LIN {X 0,Y 560.562,Z 1121.006,A -85,B 0,C 180,E1 21527.974,E2 21527.974} C_VEL
LIN {X 0,Y 560.296,Z 1132.318,A -85,B 0,C 180,E1 21525.845,E2 21525.845} C_VEL
LIN {X 0,Y 560.127,Z 1141.995,A -85,B 0,C 180,E1 21523.734,E2 21523.734} C_VEL
LIN {X 0,Y 560.015,Z 1150.716,A -85,B 0,C 180,E1 21521.425,E2 21521.425} C_VEL
LIN {X 0,Y 559.955,Z 1157.475,A -85,B 0,C 180,E1 21519.248,E2 21519.248} C_VEL
LIN {X 0,Y 559.899,Z 1162.84,A -85,B 0,C 180,E1 21516.975,E2 21516.975} C_VEL
LIN {X 0,Y 559.906,Z 1166.595,A -85,B 0,C 180,E1 21514.815,E2 21514.815} C_VEL
LIN {X 0,Y 559.915,Z 1169.055,A -85,B 0,C 180,E1 21512.456,E2 21512.456} C_VEL
LIN {X 0,Y 559.892,Z 1169.939,A -85,B 0,C 180,E1 21510.307,E2 21510.307} C_VEL
LIN {X 0,Y 559.911,Z 1169.324,A -85,B 0,C 180,E1 21507.953,E2 21507.953} C_VEL
LIN {X 0,Y 559.914,Z 1167.276,A -85,B 0,C 180,E1 21505.699,E2 21505.699} C_VEL
LIN {X 0,Y 559.914,Z 1163.461,A -85,B 0,C 180,E1 21503.334,E2 21503.334} C_VEL
LIN {X 0,Y 559.955,Z 1158.551,A -85,B 0,C 180,E1 21501.167,E2 21501.167} C_VEL
LIN {X 0,Y 560,Z 1151.764,A -85,B 0,C 180,E1 21498.882,E2 21498.882} C_VEL
LIN {X 0,Y 560.097,Z 1144.109,A -85,B 0,C 180,E1 21496.791,E2 21496.791} C_VEL
LIN {X 0,Y 560.276,Z 1133.883,A -85,B 0,C 180,E1 21494.473,E2 21494.473} C_VEL
LIN {X 0,Y 560.534,Z 1122.819,A -85,B 0,C 180,E1 21492.348,E2 21492.348} C_VEL
LIN {X 0,Y 560.864,Z 1109.753,A -85,B 0,C 180,E1 21490.201,E2 21490.201} C_VEL
LIN {X 0,Y 561.293,Z 1095.338,A -85,B 0,C 180,E1 21488.137,E2 21488.137} C_VEL
LIN {X 0,Y 561.795,Z 1079.942,A -85,B 0,C 180,E1 21486.227,E2 21486.227} C_VEL
LIN {X 0,Y 562.438,Z 1062.115,A -85,B 0,C 180,E1 21484.293,E2 21484.293} C_VEL
LIN {X 0,Y 563.12,Z 1044.253,A -85,B 0,C 180,E1 21482.595,E2 21482.595} C_VEL
LIN {X 0,Y 563.844,Z 1025.338,A -85,B 0,C 180,E1 21481.046,E2 21481.046} C_VEL
LIN {X 0,Y 564.61,Z 1004.603,A -85,B 0,C 180,E1 21479.571,E2 21479.571} C_VEL
LIN {X 0,Y 565.354,Z 984.83,A -85,B 0,C 180,E1 21478.374,E2 21478.374} C_VEL
LIN {X 0,Y 566.073,Z 962.172,A -85,B 0,C 180,E1 21477.22,E2 21477.22} C_VEL
LIN {X 0,Y 566.732,Z 941.505,A -85,B 0,C 180,E1 21476.36,E2 21476.36} C_VEL
LIN {X 0,Y 567.278,Z 918.342,A -85,B 0,C 180,E1 21475.6,E2 21475.6} C_VEL
LIN {X 0,Y 567.741,Z 896.292,A -85,B 0,C 180,E1 21475.062,E2 21475.062} C_VEL
LIN {X 0,Y 568.079,Z 859.915,A -85,B 0,C 180,E1 21474.482,E2 21474.482} C_VEL
LIN {X 0,Y 569.548,Z 649.859,A -85,B 0,C 180,E1 21471.336,E2 21471.336} C_VEL
LIN {X 0,Y 570.107,Z 551.64,A -85,B 0,C 180,E1 21469.813,E2 21469.813} C_VEL
LIN {X 0,Y 568.373,Z 542.27,A -85,B 0,C 180,E1 21469.502,E2 21469.502} C_VEL
LIN {X 0,Y 568.462,Z 530.87,A -85,B 0,C 180,E1 21468.749,E2 21468.749} C_VEL
LIN {X 0,Y 561.578,Z 516.737,A -85,B 0,C 180,E1 21467.146,E2 21467.146} C_VEL
LIN {X 0,Y 560.294,Z 513.438,A -85,B 0,C 180,E1 21466.726,E2 21466.726} C_VEL
LIN {X 0,Y 560.28,Z 513.252,A -85,B 0,C 180,E1 21463.397,E2 21463.397} C_VEL
LIN {X 0,Y 560.273,Z 513.252,A -85,B 0,C 180,E1 21459.975,E2 21459.975} C_VEL
LIN {X 0,Y 560.264,Z 513.243,A -85,B 0,C 180,E1 21456.715,E2 21456.715} C_VEL
LIN {X 0,Y 560.267,Z 513.249,A -85,B 0,C 180,E1 21453.466,E2 21453.466} C_VEL
LIN {X 0,Y 560.261,Z 513.255,A -85,B 0,C 180,E1 21450.216,E2 21450.216} C_VEL
LIN {X 0,Y 560.264,Z 513.249,A -85,B 0,C 180,E1 21446.955,E2 21446.955} C_VEL
LIN {X 0,Y 560.265,Z 513.258,A -85,B 0,C 180,E1 21443.674,E2 21443.674} C_VEL
LIN {X 0,Y 560.269,Z 513.249,A -85,B 0,C 180,E1 21440.365,E2 21440.365} C_VEL
LIN {X 0,Y 560.277,Z 513.251,A -85,B 0,C 180,E1 21436.911,E2 21436.911} C_VEL
LIN {X 0,Y 560.27,Z 513.247,A -85,B 0,C 180,E1 21433.52,E2 21433.52} C_VEL
LIN {X 0,Y 560.262,Z 513.247,A -85,B 0,C 180,E1 21430.176,E2 21430.176} C_VEL
LIN {X 0,Y 560.264,Z 513.248,A -85,B 0,C 180,E1 21426.867,E2 21426.867} C_VEL
LIN {X 0,Y 560.263,Z 513.25,A -85,B 0,C 180,E1 21423.581,E2 21423.581} C_VEL
LIN {X 0,Y 560.277,Z 513.258,A -85,B 0,C 180,E1 21420.204,E2 21420.204} C_VEL
LIN {X 0,Y 560.278,Z 513.25,A -85,B 0,C 180,E1 21416.726,E2 21416.726} C_VEL
LIN {X 0,Y 560.261,Z 513.254,A -85,B 0,C 180,E1 21413.338,E2 21413.338} C_VEL
LIN {X 0,Y 560.268,Z 513.255,A -85,B 0,C 180,E1 21410.031,E2 21410.031} C_VEL
LIN {X 0,Y 560.258,Z 513.247,A -85,B 0,C 180,E1 21406.795,E2 21406.795} C_VEL
LIN {X 0,Y 560.27,Z 513.258,A -85,B 0,C 180,E1 21403.516,E2 21403.516} C_VEL
LIN {X 0,Y 560.264,Z 513.244,A -85,B 0,C 180,E1 21400.179,E2 21400.179} C_VEL
LIN {X 0,Y 560.278,Z 513.256,A -85,B 0,C 180,E1 21396.772,E2 21396.772} C_VEL
LIN {X 0,Y 560.255,Z 513.251,A -85,B 0,C 180,E1 21396.282,E2 21396.282} C_VEL
LIN {X 0,Y 559.277,Z 513.372,A -85,B 0,C 180,E1 21395.494,E2 21395.494} C_VEL
LIN {X 0,Y 552.874,Z 514.168,A -85,B 0,C 180,E1 21393.282,E2 21393.282} C_VEL
LIN {X 0,Y 552.338,Z 514.243,A -85,B 0,C 180,E1 21392.706,E2 21392.706} C_VEL
LIN {X 0,Y 552.341,Z 514.229,A -85,B 0,C 180,E1 21389.301,E2 21389.301} C_VEL
LIN {X 0,Y 552.324,Z 514.245,A -85,B 0,C 180,E1 21385.987,E2 21385.987} C_VEL
LIN {X 0,Y 552.334,Z 514.241,A -85,B 0,C 180,E1 21382.627,E2 21382.627} C_VEL
LIN {X 0,Y 552.314,Z 514.238,A -85,B 0,C 180,E1 21379.329,E2 21379.329} C_VEL
LIN {X 0,Y 552.335,Z 514.233,A -85,B 0,C 180,E1 21375.962,E2 21375.962} C_VEL
LIN {X 0,Y 552.323,Z 514.225,A -85,B 0,C 180,E1 21372.613,E2 21372.613} C_VEL
LIN {X 0,Y 552.388,Z 514.576,A -85,B 0,C 180,E1 21371.593,E2 21371.593} C_VEL
LIN {X 0,Y 554.03,Z 518.332,A -85,B 0,C 180,E1 21371.109,E2 21371.109} C_VEL
LIN {X 0,Y 560.868,Z 533.617,A -85,B 0,C 180,E1 21369.368,E2 21369.368} C_VEL
LIN {X 0,Y 559.531,Z 581.004,A -85,B 0,C 180,E1 21366.127,E2 21366.127} C_VEL
LIN {X 0,Y 559.41,Z 590.555,A -85,B 0,C 180,E1 21365.522,E2 21365.522} C_VEL
LIN {X 0,Y 561.19,Z 601.495,A -85,B 0,C 180,E1 21365.221,E2 21365.221} C_VEL
LIN {X 0,Y 559.53,Z 831.551,A -85,B 0,C 180,E1 21361.866,E2 21361.866} C_VEL
LIN {X 0,Y 559.039,Z 897.029,A -85,B 0,C 180,E1 21360.896,E2 21360.896} C_VEL
LIN {X 0,Y 558.577,Z 918.635,A -85,B 0,C 180,E1 21360.381,E2 21360.381} C_VEL
LIN {X 0,Y 558.024,Z 940.668,A -85,B 0,C 180,E1 21359.655,E2 21359.655} C_VEL
LIN {X 0,Y 557.432,Z 961.155,A -85,B 0,C 180,E1 21358.79,E2 21358.79} C_VEL
LIN {X 0,Y 556.733,Z 980.474,A -85,B 0,C 180,E1 21357.778,E2 21357.778} C_VEL
LIN {X 0,Y 555.975,Z 1001.01,A -85,B 0,C 180,E1 21356.487,E2 21356.487} C_VEL
LIN {X 0,Y 555.267,Z 1019.082,A -85,B 0,C 180,E1 21355.148,E2 21355.148} C_VEL
LIN {X 0,Y 554.564,Z 1036.919,A -85,B 0,C 180,E1 21353.594,E2 21353.594} C_VEL
LIN {X 0,Y 553.926,Z 1053.575,A -85,B 0,C 180,E1 21351.907,E2 21351.907} C_VEL
LIN {X 0,Y 553.35,Z 1069.662,A -85,B 0,C 180,E1 21350.016,E2 21350.016} C_VEL
LIN {X 0,Y 552.9,Z 1083.542,A -85,B 0,C 180,E1 21348.122,E2 21348.122} C_VEL
LIN {X 0,Y 552.547,Z 1095.699,A -85,B 0,C 180,E1 21346.181,E2 21346.181} C_VEL
LIN {X 0,Y 552.274,Z 1107.096,A -85,B 0,C 180,E1 21344.04,E2 21344.04} C_VEL
LIN {X 0,Y 552.098,Z 1116.58,A -85,B 0,C 180,E1 21341.915,E2 21341.915} C_VEL
LIN {X 0,Y 551.991,Z 1124.218,A -85,B 0,C 180,E1 21339.808,E2 21339.808} C_VEL
LIN {X 0,Y 551.933,Z 1130.536,A -85,B 0,C 180,E1 21337.599,E2 21337.599} C_VEL
LIN {X 0,Y 551.913,Z 1135.247,A -85,B 0,C 180,E1 21335.406,E2 21335.406} C_VEL
LIN {X 0,Y 551.909,Z 1138.236,A -85,B 0,C 180,E1 21333.219,E2 21333.219} C_VEL
LIN {X 0,Y 551.906,Z 1139.795,A -85,B 0,C 180,E1 21330.934,E2 21330.934} C_VEL
LIN {X 0,Y 551.91,Z 1139.747,A -85,B 0,C 180,E1 21328.754,E2 21328.754} C_VEL
LIN {X 0,Y 551.914,Z 1138.102,A -85,B 0,C 180,E1 21326.566,E2 21326.566} C_VEL
LIN {X 0,Y 551.922,Z 1135.016,A -85,B 0,C 180,E1 21324.386,E2 21324.386} C_VEL
LIN {X 0,Y 551.936,Z 1130.443,A -85,B 0,C 180,E1 21322.272,E2 21322.272} C_VEL
LIN {X 0,Y 551.999,Z 1123.827,A -85,B 0,C 180,E1 21319.986,E2 21319.986} C_VEL
LIN {X 0,Y 552.112,Z 1116.11,A -85,B 0,C 180,E1 21317.873,E2 21317.873} C_VEL
LIN {X 0,Y 552.292,Z 1106.494,A -85,B 0,C 180,E1 21315.746,E2 21315.746} C_VEL
LIN {X 0,Y 552.57,Z 1094.958,A -85,B 0,C 180,E1 21313.604,E2 21313.604} C_VEL
LIN {X 0,Y 552.928,Z 1082.692,A -85,B 0,C 180,E1 21311.661,E2 21311.661} C_VEL
LIN {X 0,Y 553.372,Z 1069.014,A -85,B 0,C 180,E1 21309.811,E2 21309.811} C_VEL
LIN {X 0,Y 553.947,Z 1053.078,A -85,B 0,C 180,E1 21307.949,E2 21307.949} C_VEL
LIN {X 0,Y 554.603,Z 1035.953,A -85,B 0,C 180,E1 21306.227,E2 21306.227} C_VEL
LIN {X 0,Y 555.316,Z 1017.95,A -85,B 0,C 180,E1 21304.671,E2 21304.671} C_VEL
LIN {X 0,Y 556.05,Z 999.031,A -85,B 0,C 180,E1 21303.286,E2 21303.286} C_VEL
LIN {X 0,Y 556.788,Z 979.033,A -85,B 0,C 180,E1 21302.05,E2 21302.05} C_VEL
LIN {X 0,Y 557.472,Z 959.341,A -85,B 0,C 180,E1 21301.036,E2 21301.036} C_VEL
LIN {X 0,Y 558.068,Z 939.628,A -85,B 0,C 180,E1 21300.216,E2 21300.216} C_VEL
LIN {X 0,Y 558.594,Z 917.254,A -85,B 0,C 180,E1 21299.491,E2 21299.491} C_VEL
LIN {X 0,Y 559.054,Z 895.666,A -85,B 0,C 180,E1 21298.991,E2 21298.991} C_VEL
LIN {X 0,Y 560.624,Z 674.56,A -85,B 0,C 180,E1 21295.764,E2 21295.764} C_VEL
LIN {X 0,Y 560.976,Z 601.536,A -85,B 0,C 180,E1 21294.674,E2 21294.674} C_VEL
LIN {X 0,Y 558.666,Z 590.554,A -85,B 0,C 180,E1 21294.306,E2 21294.306} C_VEL
LIN {X 0,Y 559.886,Z 549.146,A -85,B 0,C 180,E1 21290.92,E2 21290.92} C_VEL
LIN {X 0,Y 560.191,Z 533.38,A -85,B 0,C 180,E1 21289.574,E2 21289.574} C_VEL
LIN {X 0,Y 553.416,Z 517.359,A -85,B 0,C 180,E1 21287.488,E2 21287.488} C_VEL
LIN {X 0,Y 552.342,Z 514.443,A -85,B 0,C 180,E1 21287.064,E2 21287.064} C_VEL
LIN {X 0,Y 552.283,Z 514.237,A -85,B 0,C 180,E1 21284.043,E2 21284.043} C_VEL
LIN {X 0,Y 552.303,Z 514.239,A -85,B 0,C 180,E1 21280.665,E2 21280.665} C_VEL
LIN {X 0,Y 552.28,Z 514.249,A -85,B 0,C 180,E1 21277.706,E2 21277.706} C_VEL
LIN {X 0,Y 552.336,Z 514.514,A -85,B 0,C 180,E1 21275.33,E2 21275.33} C_VEL
LIN {X 0,Y 556.826,Z 528.593,A -85,B 0,C 180,E1 21273.943,E2 21273.943} C_VEL
LIN {X 0,Y 556.497,Z 566.554,A -85,B 0,C 180,E1 21271.015,E2 21271.015} C_VEL
LIN {X 0,Y 555.991,Z 605.609,A -85,B 0,C 180,E1 21267.993,E2 21267.993} C_VEL
LIN {X 0,Y 555.136,Z 647.932,A -85,B 0,C 180,E1 21264.7,E2 21264.7} C_VEL
LIN {X 0,Y 554.341,Z 692.274,A -85,B 0,C 180,E1 21261.312,E2 21261.312} C_VEL
LIN {X 0,Y 554.138,Z 705.669,A -85,B 0,C 180,E1 21260.336,E2 21260.336} C_VEL
LIN {X 0,Y 554.992,Z 713.85,A -85,B 0,C 180,E1 21260.192,E2 21260.192} C_VEL
LIN {X 0,Y 554.361,Z 876.056,A -85,B 0,C 180,E1 21258.008,E2 21258.008} C_VEL
LIN {X 0,Y 554.144,Z 893.538,A -85,B 0,C 180,E1 21257.571,E2 21257.571} C_VEL
LIN {X 0,Y 553.859,Z 910.683,A -85,B 0,C 180,E1 21256.946,E2 21256.946} C_VEL
LIN {X 0,Y 553.556,Z 926.795,A -85,B 0,C 180,E1 21256.151,E2 21256.151} C_VEL
LIN {X 0,Y 553.207,Z 942.641,A -85,B 0,C 180,E1 21255.145,E2 21255.145} C_VEL
LIN {X 0,Y 552.864,Z 957.964,A -85,B 0,C 180,E1 21253.918,E2 21253.918} C_VEL
LIN {X 0,Y 552.575,Z 970.819,A -85,B 0,C 180,E1 21252.647,E2 21252.647} C_VEL
LIN {X 0,Y 552.341,Z 982.209,A -85,B 0,C 180,E1 21251.274,E2 21251.274} C_VEL
LIN {X 0,Y 552.158,Z 992.869,A -85,B 0,C 180,E1 21249.695,E2 21249.695} C_VEL
LIN {X 0,Y 552.03,Z 1001.869,A -85,B 0,C 180,E1 21248.017,E2 21248.017} C_VEL
LIN {X 0,Y 551.96,Z 1008.816,A -85,B 0,C 180,E1 21246.344,E2 21246.344} C_VEL
LIN {X 0,Y 551.925,Z 1014.226,A -85,B 0,C 180,E1 21244.572,E2 21244.572} C_VEL
LIN {X 0,Y 551.915,Z 1017.967,A -85,B 0,C 180,E1 21242.7,E2 21242.7} C_VEL
LIN {X 0,Y 551.914,Z 1019.781,A -85,B 0,C 180,E1 21240.831,E2 21240.831} C_VEL
LIN {X 0,Y 551.915,Z 1019.746,A -85,B 0,C 180,E1 21239.066,E2 21239.066} C_VEL
LIN {X 0,Y 551.915,Z 1018.103,A -85,B 0,C 180,E1 21237.301,E2 21237.301} C_VEL
LIN {X 0,Y 551.925,Z 1014.451,A -85,B 0,C 180,E1 21235.428,E2 21235.428} C_VEL
LIN {X 0,Y 551.955,Z 1009.461,A -85,B 0,C 180,E1 21233.761,E2 21233.761} C_VEL
LIN {X 0,Y 552.02,Z 1002.789,A -85,B 0,C 180,E1 21232.088,E2 21232.088} C_VEL
LIN {X 0,Y 552.14,Z 994.047,A -85,B 0,C 180,E1 21230.41,E2 21230.41} C_VEL
LIN {X 0,Y 552.317,Z 983.658,A -85,B 0,C 180,E1 21228.831,E2 21228.831} C_VEL
LIN {X 0,Y 552.564,Z 971.117,A -85,B 0,C 180,E1 21227.3,E2 21227.3} C_VEL
LIN {X 0,Y 552.818,Z 959.469,A -85,B 0,C 180,E1 21226.135,E2 21226.135} C_VEL
LIN {X 0,Y 553.134,Z 946.112,A -85,B 0,C 180,E1 21225.02,E2 21225.02} C_VEL
LIN {X 0,Y 553.47,Z 930.113,A -85,B 0,C 180,E1 21223.955,E2 21223.955} C_VEL
LIN {X 0,Y 553.749,Z 915.956,A -85,B 0,C 180,E1 21223.208,E2 21223.208} C_VEL
LIN {X 0,Y 554.051,Z 900.589,A -85,B 0,C 180,E1 21222.569,E2 21222.569} C_VEL
LIN {X 0,Y 554.278,Z 883.504,A -85,B 0,C 180,E1 21222.066,E2 21222.066} C_VEL
LIN {X 0,Y 554.42,Z 865.876,A -85,B 0,C 180,E1 21221.739,E2 21221.739} C_VEL
LIN {X 0,Y 554.815,Z 710.464,A -85,B 0,C 180,E1 21219.665,E2 21219.665} C_VEL
LIN {X 0,Y 554.077,Z 704.577,A -85,B 0,C 180,E1 21219.522,E2 21219.522} C_VEL
LIN {X 0,Y 554.903,Z 660.003,A -85,B 0,C 180,E1 21216.139,E2 21216.139} C_VEL
LIN {X 0,Y 555.761,Z 617.071,A -85,B 0,C 180,E1 21212.809,E2 21212.809} C_VEL
LIN {X 0,Y 556.004,Z 585.332,A -85,B 0,C 180,E1 21210.438,E2 21210.438} C_VEL
LIN {X 0,Y 555.825,Z 557.018,A -85,B 0,C 180,E1 21208.435,E2 21208.435} C_VEL
LIN {X 0,Y 555.246,Z 527.459,A -85,B 0,C 180,E1 21206.486,E2 21206.486} C_VEL
LIN {X 0,Y 554.798,Z 524.469,A -85,B 0,C 180,E1 21206.284,E2 21206.284} C_VEL
LIN {X 0,Y 552.369,Z 514.601,A -85,B 0,C 180,E1 21205.568,E2 21205.568} C_VEL
LIN {X 0,Y 552.343,Z 514.249,A -85,B 0,C 180,E1 21205.088,E2 21205.088} C_VEL
LIN {X 0,Y 552.318,Z 514.245,A -85,B 0,C 180,E1 21201.749,E2 21201.749} C_VEL
LIN {X 0,Y 552.325,Z 514.244,A -85,B 0,C 180,E1 21198.367,E2 21198.367} C_VEL
LIN {X 0,Y 552.319,Z 514.23,A -85,B 0,C 180,E1 21195.058,E2 21195.058} C_VEL
LIN {X 0,Y 552.388,Z 514.56,A -85,B 0,C 180,E1 21194.396,E2 21194.396} C_VEL
LIN {X 0,Y 553.864,Z 518.049,A -85,B 0,C 180,E1 21193.922,E2 21193.922} C_VEL
LIN {X 0,Y 561.374,Z 535.018,A -85,B 0,C 180,E1 21191.769,E2 21191.769} C_VEL
LIN {X 0,Y 561.249,Z 543.948,A -85,B 0,C 180,E1 21191.09,E2 21191.09} C_VEL
LIN {X 0,Y 564.108,Z 557.393,A -85,B 0,C 180,E1 21190.61,E2 21190.61} C_VEL
LIN {X 0,Y 562.326,Z 765.247,A -85,B 0,C 180,E1 21187.415,E2 21187.415} C_VEL
LIN {X 0,Y 561.248,Z 892.082,A -85,B 0,C 180,E1 21185.487,E2 21185.487} C_VEL
LIN {X 0,Y 560.694,Z 915.746,A -85,B 0,C 180,E1 21184.939,E2 21184.939} C_VEL
LIN {X 0,Y 560.122,Z 937.778,A -85,B 0,C 180,E1 21184.241,E2 21184.241} C_VEL
LIN {X 0,Y 559.344,Z 959.681,A -85,B 0,C 180,E1 21183.345,E2 21183.345} C_VEL
LIN {X 0,Y 558.545,Z 980.784,A -85,B 0,C 180,E1 21182.3,E2 21182.3} C_VEL
LIN {X 0,Y 557.68,Z 1001.047,A -85,B 0,C 180,E1 21181.088,E2 21181.088} C_VEL
LIN {X 0,Y 556.795,Z 1020.931,A -85,B 0,C 180,E1 21179.711,E2 21179.711} C_VEL
LIN {X 0,Y 555.953,Z 1039.504,A -85,B 0,C 180,E1 21178.208,E2 21178.208} C_VEL
LIN {X 0,Y 555.077,Z 1058.792,A -85,B 0,C 180,E1 21176.418,E2 21176.418} C_VEL
LIN {X 0,Y 554.366,Z 1075.661,A -85,B 0,C 180,E1 21174.622,E2 21174.622} C_VEL
LIN {X 0,Y 553.688,Z 1091.994,A -85,B 0,C 180,E1 21172.621,E2 21172.621} C_VEL
LIN {X 0,Y 553.14,Z 1106.919,A -85,B 0,C 180,E1 21170.529,E2 21170.529} C_VEL
LIN {X 0,Y 552.722,Z 1119.734,A -85,B 0,C 180,E1 21168.456,E2 21168.456} C_VEL
LIN {X 0,Y 552.396,Z 1131.799,A -85,B 0,C 180,E1 21166.185,E2 21166.185} C_VEL
LIN {X 0,Y 552.203,Z 1141.076,A -85,B 0,C 180,E1 21164.149,E2 21164.149} C_VEL
LIN {X 0,Y 552.051,Z 1150.341,A -85,B 0,C 180,E1 21161.704,E2 21161.704} C_VEL
LIN {X 0,Y 551.951,Z 1156.868,A -85,B 0,C 180,E1 21159.594,E2 21159.594} C_VEL
LIN {X 0,Y 551.902,Z 1162.634,A -85,B 0,C 180,E1 21157.181,E2 21157.181} C_VEL
LIN {X 0,Y 551.913,Z 1166.276,A -85,B 0,C 180,E1 21155.093,E2 21155.093} C_VEL
LIN {X 0,Y 551.91,Z 1168.988,A -85,B 0,C 180,E1 21152.596,E2 21152.596} C_VEL
LIN {X 0,Y 551.884,Z 1169.895,A -85,B 0,C 180,E1 21150.519,E2 21150.519} C_VEL
LIN {X 0,Y 551.908,Z 1169.391,A -85,B 0,C 180,E1 21148.027,E2 21148.027} C_VEL
LIN {X 0,Y 551.917,Z 1167.503,A -85,B 0,C 180,E1 21145.844,E2 21145.844} C_VEL
LIN {X 0,Y 551.916,Z 1163.667,A -85,B 0,C 180,E1 21143.342,E2 21143.342} C_VEL
LIN {X 0,Y 551.96,Z 1159.061,A -85,B 0,C 180,E1 21141.248,E2 21141.248} C_VEL
LIN {X 0,Y 552.018,Z 1152.119,A -85,B 0,C 180,E1 21138.825,E2 21138.825} C_VEL
LIN {X 0,Y 552.129,Z 1144.519,A -85,B 0,C 180,E1 21136.704,E2 21136.704} C_VEL
LIN {X 0,Y 552.342,Z 1134.4,A -85,B 0,C 180,E1 21134.352,E2 21134.352} C_VEL
LIN {X 0,Y 552.639,Z 1123.402,A -85,B 0,C 180,E1 21132.196,E2 21132.196} C_VEL
LIN {X 0,Y 553.038,Z 1110.464,A -85,B 0,C 180,E1 21130.019,E2 21130.019} C_VEL
LIN {X 0,Y 553.551,Z 1096.068,A -85,B 0,C 180,E1 21127.912,E2 21127.912} C_VEL
LIN {X 0,Y 554.162,Z 1080.254,A -85,B 0,C 180,E1 21125.917,E2 21125.917} C_VEL
LIN {X 0,Y 554.942,Z 1062.116,A -85,B 0,C 180,E1 21123.92,E2 21123.92} C_VEL
LIN {X 0,Y 555.763,Z 1043.896,A -85,B 0,C 180,E1 21122.169,E2 21122.169} C_VEL
LIN {X 0,Y 556.617,Z 1024.907,A -85,B 0,C 180,E1 21120.599,E2 21120.599} C_VEL
LIN {X 0,Y 557.56,Z 1003.716,A -85,B 0,C 180,E1 21119.084,E2 21119.084} C_VEL
LIN {X 0,Y 558.416,Z 983.884,A -85,B 0,C 180,E1 21117.877,E2 21117.877} C_VEL
LIN {X 0,Y 559.233,Z 962.234,A -85,B 0,C 180,E1 21116.77,E2 21116.77} C_VEL
LIN {X 0,Y 559.996,Z 941.503,A -85,B 0,C 180,E1 21115.9,E2 21115.9} C_VEL
LIN {X 0,Y 560.63,Z 918.219,A -85,B 0,C 180,E1 21115.13,E2 21115.13} C_VEL
LIN {X 0,Y 561.192,Z 895.804,A -85,B 0,C 180,E1 21114.581,E2 21114.581} C_VEL
LIN {X 0,Y 561.6,Z 855.786,A -85,B 0,C 180,E1 21113.945,E2 21113.945} C_VEL
LIN {X 0,Y 563.331,Z 646.028,A -85,B 0,C 180,E1 21110.767,E2 21110.767} C_VEL
LIN {X 0,Y 563.997,Z 553.429,A -85,B 0,C 180,E1 21109.316,E2 21109.316} C_VEL
LIN {X 0,Y 561.94,Z 542.168,A -85,B 0,C 180,E1 21108.935,E2 21108.935} C_VEL
LIN {X 0,Y 561.962,Z 534.582,A -85,B 0,C 180,E1 21108.421,E2 21108.421} C_VEL
LIN {X 0,Y 553.971,Z 518.181,A -85,B 0,C 180,E1 21106.515,E2 21106.515} C_VEL
LIN {X 0,Y 552.379,Z 514.586,A -85,B 0,C 180,E1 21106.062,E2 21106.062} C_VEL
LIN {X 0,Y 552.325,Z 514.23,A -85,B 0,C 180,E1 21105.204,E2 21105.204} C_VEL
LIN {X 0,Y 552.329,Z 514.241,A -85,B 0,C 180,E1 21101.911,E2 21101.911} C_VEL
LIN {X 0,Y 552.323,Z 514.248,A -85,B 0,C 180,E1 21098.552,E2 21098.552} C_VEL
LIN {X 0,Y 552.331,Z 514.245,A -85,B 0,C 180,E1 21095.271,E2 21095.271} C_VEL
LIN {X 0,Y 552.332,Z 514.234,A -85,B 0,C 180,E1 21091.896,E2 21091.896} C_VEL
LIN {X 0,Y 552.336,Z 514.238,A -85,B 0,C 180,E1 21088.43,E2 21088.43} C_VEL
LIN {X 0,Y 552.328,Z 514.248,A -85,B 0,C 180,E1 21085.062,E2 21085.062} C_VEL
LIN {X 0,Y 552.325,Z 514.232,A -85,B 0,C 180,E1 21081.771,E2 21081.771} C_VEL
LIN {X 0,Y 552.327,Z 514.244,A -85,B 0,C 180,E1 21078.453,E2 21078.453} C_VEL
LIN {X 0,Y 552.328,Z 514.23,A -85,B 0,C 180,E1 21075.11,E2 21075.11} C_VEL
LIN {X 0,Y 552.339,Z 514.24,A -85,B 0,C 180,E1 21071.668,E2 21071.668} C_VEL
LIN {X 0,Y 552.326,Z 514.232,A -85,B 0,C 180,E1 21068.222,E2 21068.222} C_VEL
LIN {X 0,Y 552.328,Z 514.244,A -85,B 0,C 180,E1 21064.88,E2 21064.88} C_VEL
LIN {X 0,Y 552.322,Z 514.244,A -85,B 0,C 180,E1 21061.556,E2 21061.556} C_VEL
LIN {X 0,Y 552.331,Z 514.246,A -85,B 0,C 180,E1 21058.236,E2 21058.236} C_VEL
LIN {X 0,Y 552.336,Z 514.24,A -85,B 0,C 180,E1 21054.807,E2 21054.807} C_VEL
LIN {X 0,Y 552.328,Z 514.248,A -85,B 0,C 180,E1 21051.358,E2 21051.358} C_VEL
LIN {X 0,Y 552.33,Z 514.234,A -85,B 0,C 180,E1 21047.984,E2 21047.984} C_VEL
LIN {X 0,Y 552.318,Z 514.245,A -85,B 0,C 180,E1 21044.674,E2 21044.674} C_VEL
LIN {X 0,Y 552.333,Z 514.234,A -85,B 0,C 180,E1 21041.312,E2 21041.312} C_VEL
LIN {X 0,Y 552.338,Z 514.241,A -85,B 0,C 180,E1 21037.881,E2 21037.881} C_VEL
LIN {X 0,Y 552.326,Z 514.234,A -85,B 0,C 180,E1 21034.479,E2 21034.479} C_VEL
LIN {X 0,Y 552.338,Z 514.243,A -85,B 0,C 180,E1 21032.706,E2 21032.706} C_VEL
LIN {X 0,Y 551.35,Z 514.375,A -85,B 0,C 180,E1 21031.907,E2 21031.907} C_VEL
LIN {X 0,Y 544.847,Z 515.163,A -85,B 0,C 180,E1 21029.605,E2 21029.605} C_VEL
LIN {X 0,Y 544.396,Z 515.217,A -85,B 0,C 180,E1 21029.079,E2 21029.079} C_VEL
LIN {X 0,Y 544.377,Z 515.231,A -85,B 0,C 180,E1 21025.743,E2 21025.743} C_VEL
LIN {X 0,Y 544.394,Z 515.232,A -85,B 0,C 180,E1 21022.427,E2 21022.427} C_VEL
LIN {X 0,Y 544.377,Z 515.227,A -85,B 0,C 180,E1 21019.166,E2 21019.166} C_VEL
LIN {X 0,Y 544.399,Z 515.219,A -85,B 0,C 180,E1 21015.739,E2 21015.739} C_VEL
LIN {X 0,Y 544.413,Z 515.335,A -85,B 0,C 180,E1 21012.379,E2 21012.379} C_VEL
LIN {X 0,Y 544.535,Z 515.993,A -85,B 0,C 180,E1 21012.225,E2 21012.225} C_VEL
LIN {X 0,Y 552.88,Z 534.192,A -85,B 0,C 180,E1 21010.014,E2 21010.014} C_VEL
LIN {X 0,Y 554.194,Z 537.39,A -85,B 0,C 180,E1 21009.66,E2 21009.66} C_VEL
LIN {X 0,Y 552.65,Z 584.849,A -85,B 0,C 180,E1 21006.38,E2 21006.38} C_VEL
LIN {X 0,Y 552.626,Z 590.599,A -85,B 0,C 180,E1 21006.026,E2 21006.026} C_VEL
LIN {X 0,Y 554.645,Z 602.933,A -85,B 0,C 180,E1 21005.678,E2 21005.678} C_VEL
LIN {X 0,Y 552.725,Z 833.51,A -85,B 0,C 180,E1 21002.277,E2 21002.277} C_VEL
LIN {X 0,Y 552.172,Z 897.066,A -85,B 0,C 180,E1 21001.323,E2 21001.323} C_VEL
LIN {X 0,Y 551.641,Z 918.695,A -85,B 0,C 180,E1 21000.803,E2 21000.803} C_VEL
LIN {X 0,Y 551.032,Z 940.353,A -85,B 0,C 180,E1 21000.084,E2 21000.084} C_VEL
LIN {X 0,Y 550.352,Z 959.947,A -85,B 0,C 180,E1 20999.256,E2 20999.256} C_VEL
LIN {X 0,Y 549.571,Z 979.496,A -85,B 0,C 180,E1 20998.231,E2 20998.231} C_VEL
LIN {X 0,Y 548.683,Z 1000.206,A -85,B 0,C 180,E1 20996.926,E2 20996.926} C_VEL
LIN {X 0,Y 547.838,Z 1019.088,A -85,B 0,C 180,E1 20995.514,E2 20995.514} C_VEL
LIN {X 0,Y 547.022,Z 1036.928,A -85,B 0,C 180,E1 20993.94,E2 20993.94} C_VEL
LIN {X 0,Y 546.285,Z 1053.274,A -85,B 0,C 180,E1 20992.264,E2 20992.264} C_VEL
LIN {X 0,Y 545.616,Z 1069.179,A -85,B 0,C 180,E1 20990.376,E2 20990.376} C_VEL
LIN {X 0,Y 545.109,Z 1082.828,A -85,B 0,C 180,E1 20988.501,E2 20988.501} C_VEL
LIN {X 0,Y 544.672,Z 1095.701,A -85,B 0,C 180,E1 20986.421,E2 20986.421} C_VEL
LIN {X 0,Y 544.349,Z 1107.1,A -85,B 0,C 180,E1 20984.249,E2 20984.249} C_VEL
LIN {X 0,Y 544.139,Z 1116.583,A -85,B 0,C 180,E1 20982.092,E2 20982.092} C_VEL
LIN {X 0,Y 544.013,Z 1124.234,A -85,B 0,C 180,E1 20979.949,E2 20979.949} C_VEL
LIN {X 0,Y 543.945,Z 1130.538,A -85,B 0,C 180,E1 20977.712,E2 20977.712} C_VEL
LIN {X 0,Y 543.918,Z 1135.248,A -85,B 0,C 180,E1 20975.485,E2 20975.485} C_VEL
LIN {X 0,Y 543.911,Z 1138.237,A -85,B 0,C 180,E1 20973.267,E2 20973.267} C_VEL
LIN {X 0,Y 543.907,Z 1139.795,A -85,B 0,C 180,E1 20970.948,E2 20970.948} C_VEL
LIN {X 0,Y 543.909,Z 1139.747,A -85,B 0,C 180,E1 20968.736,E2 20968.736} C_VEL
LIN {X 0,Y 543.912,Z 1138.109,A -85,B 0,C 180,E1 20966.522,E2 20966.522} C_VEL
LIN {X 0,Y 543.926,Z 1135.015,A -85,B 0,C 180,E1 20964.303,E2 20964.303} C_VEL
LIN {X 0,Y 543.945,Z 1130.498,A -85,B 0,C 180,E1 20962.182,E2 20962.182} C_VEL
LIN {X 0,Y 544.023,Z 1123.825,A -85,B 0,C 180,E1 20959.838,E2 20959.838} C_VEL
LIN {X 0,Y 544.155,Z 1116.108,A -85,B 0,C 180,E1 20957.693,E2 20957.693} C_VEL
LIN {X 0,Y 544.37,Z 1106.492,A -85,B 0,C 180,E1 20955.535,E2 20955.535} C_VEL
LIN {X 0,Y 544.695,Z 1094.953,A -85,B 0,C 180,E1 20953.36,E2 20953.36} C_VEL
LIN {X 0,Y 545.115,Z 1082.686,A -85,B 0,C 180,E1 20951.388,E2 20951.388} C_VEL
LIN {X 0,Y 545.64,Z 1068.556,A -85,B 0,C 180,E1 20949.453,E2 20949.453} C_VEL
LIN {X 0,Y 546.297,Z 1053.071,A -85,B 0,C 180,E1 20947.623,E2 20947.623} C_VEL
LIN {X 0,Y 547.061,Z 1036.068,A -85,B 0,C 180,E1 20945.89,E2 20945.89} C_VEL
LIN {X 0,Y 547.893,Z 1018.099,A -85,B 0,C 180,E1 20944.315,E2 20944.315} C_VEL
LIN {X 0,Y 548.732,Z 999.017,A -85,B 0,C 180,E1 20942.901,E2 20942.901} C_VEL
LIN {X 0,Y 549.59,Z 979.019,A -85,B 0,C 180,E1 20941.651,E2 20941.651} C_VEL
LIN {X 0,Y 550.37,Z 959.328,A -85,B 0,C 180,E1 20940.626,E2 20940.626} C_VEL
LIN {X 0,Y 551.069,Z 939.532,A -85,B 0,C 180,E1 20939.795,E2 20939.795} C_VEL
LIN {X 0,Y 551.667,Z 917.227,A -85,B 0,C 180,E1 20939.066,E2 20939.066} C_VEL
LIN {X 0,Y 552.19,Z 895.506,A -85,B 0,C 180,E1 20938.559,E2 20938.559} C_VEL
LIN {X 0,Y 553.992,Z 676.291,A -85,B 0,C 180,E1 20935.323,E2 20935.323} C_VEL
LIN {X 0,Y 554.445,Z 603.243,A -85,B 0,C 180,E1 20934.222,E2 20934.222} C_VEL
LIN {X 0,Y 551.776,Z 590.542,A -85,B 0,C 180,E1 20933.791,E2 20933.791} C_VEL
LIN {X 0,Y 553.194,Z 549.087,A -85,B 0,C 180,E1 20930.351,E2 20930.351} C_VEL
LIN {X 0,Y 553.485,Z 537.023,A -85,B 0,C 180,E1 20929.297,E2 20929.297} C_VEL
LIN {X 0,Y 545.912,Z 519.09,A -85,B 0,C 180,E1 20926.908,E2 20926.908} C_VEL
LIN {X 0,Y 544.369,Z 515.432,A -85,B 0,C 180,E1 20926.354,E2 20926.354} C_VEL
LIN {X 0,Y 544.401,Z 515.195,A -85,B 0,C 180,E1 20923.185,E2 20923.185} C_VEL
LIN {X 0,Y 544.338,Z 515.24,A -85,B 0,C 180,E1 20920.007,E2 20920.007} C_VEL
LIN {X 0,Y 544.399,Z 515.236,A -85,B 0,C 180,E1 20916.78,E2 20916.78} C_VEL
LIN {X 0,Y 544.374,Z 515.498,A -85,B 0,C 180,E1 20915.725,E2 20915.725} C_VEL
LIN {X 0,Y 549.498,Z 531.756,A -85,B 0,C 180,E1 20914.115,E2 20914.115} C_VEL
LIN {X 0,Y 549.092,Z 569.95,A -85,B 0,C 180,E1 20911.147,E2 20911.147} C_VEL
LIN {X 0,Y 548.453,Z 611.185,A -85,B 0,C 180,E1 20907.939,E2 20907.939} C_VEL
LIN {X 0,Y 547.56,Z 652.303,A -85,B 0,C 180,E1 20904.719,E2 20904.719} C_VEL
LIN {X 0,Y 546.659,Z 695.918,A -85,B 0,C 180,E1 20901.345,E2 20901.345} C_VEL
LIN {X 0,Y 546.508,Z 705.718,A -85,B 0,C 180,E1 20900.632,E2 20900.632} C_VEL
LIN {X 0,Y 547.482,Z 714.768,A -85,B 0,C 180,E1 20900.47,E2 20900.47} C_VEL
LIN {X 0,Y 546.753,Z 876.08,A -85,B 0,C 180,E1 20898.268,E2 20898.268} C_VEL
LIN {X 0,Y 546.506,Z 893.434,A -85,B 0,C 180,E1 20897.828,E2 20897.828} C_VEL
LIN {X 0,Y 546.183,Z 910.571,A -85,B 0,C 180,E1 20897.197,E2 20897.197} C_VEL
LIN {X 0,Y 545.827,Z 926.803,A -85,B 0,C 180,E1 20896.386,E2 20896.386} C_VEL
LIN {X 0,Y 545.419,Z 942.697,A -85,B 0,C 180,E1 20895.363,E2 20895.363} C_VEL
LIN {X 0,Y 545.027,Z 957.976,A -85,B 0,C 180,E1 20894.122,E2 20894.122} C_VEL
LIN {X 0,Y 544.693,Z 970.823,A -85,B 0,C 180,E1 20892.833,E2 20892.833} C_VEL
LIN {X 0,Y 544.418,Z 982.214,A -85,B 0,C 180,E1 20891.441,E2 20891.441} C_VEL
LIN {X 0,Y 544.203,Z 992.877,A -85,B 0,C 180,E1 20889.839,E2 20889.839} C_VEL
LIN {X 0,Y 544.051,Z 1001.872,A -85,B 0,C 180,E1 20888.136,E2 20888.136} C_VEL
LIN {X 0,Y 543.968,Z 1008.816,A -85,B 0,C 180,E1 20886.438,E2 20886.438} C_VEL
LIN {X 0,Y 543.928,Z 1014.229,A -85,B 0,C 180,E1 20884.64,E2 20884.64} C_VEL
LIN {X 0,Y 543.916,Z 1017.971,A -85,B 0,C 180,E1 20882.74,E2 20882.74} C_VEL
LIN {X 0,Y 543.914,Z 1019.781,A -85,B 0,C 180,E1 20880.843,E2 20880.843} C_VEL
LIN {X 0,Y 543.916,Z 1019.739,A -85,B 0,C 180,E1 20879.052,E2 20879.052} C_VEL
LIN {X 0,Y 543.915,Z 1018.105,A -85,B 0,C 180,E1 20877.261,E2 20877.261} C_VEL
LIN {X 0,Y 543.927,Z 1014.451,A -85,B 0,C 180,E1 20875.361,E2 20875.361} C_VEL
LIN {X 0,Y 543.962,Z 1009.455,A -85,B 0,C 180,E1 20873.668,E2 20873.668} C_VEL
LIN {X 0,Y 544.04,Z 1002.787,A -85,B 0,C 180,E1 20871.971,E2 20871.971} C_VEL
LIN {X 0,Y 544.181,Z 994.043,A -85,B 0,C 180,E1 20870.268,E2 20870.268} C_VEL
LIN {X 0,Y 544.388,Z 983.653,A -85,B 0,C 180,E1 20868.667,E2 20868.667} C_VEL
LIN {X 0,Y 544.667,Z 971.598,A -85,B 0,C 180,E1 20867.167,E2 20867.167} C_VEL
LIN {X 0,Y 544.959,Z 960.027,A -85,B 0,C 180,E1 20865.985,E2 20865.985} C_VEL
LIN {X 0,Y 545.294,Z 947.436,A -85,B 0,C 180,E1 20864.908,E2 20864.908} C_VEL
LIN {X 0,Y 545.704,Z 931.305,A -85,B 0,C 180,E1 20863.792,E2 20863.792} C_VEL
LIN {X 0,Y 546.027,Z 917.055,A -85,B 0,C 180,E1 20863.019,E2 20863.019} C_VEL
LIN {X 0,Y 546.364,Z 902.016,A -85,B 0,C 180,E1 20862.37,E2 20862.37} C_VEL
LIN {X 0,Y 546.642,Z 884.339,A -85,B 0,C 180,E1 20861.829,E2 20861.829} C_VEL
LIN {X 0,Y 546.817,Z 867.081,A -85,B 0,C 180,E1 20861.494,E2 20861.494} C_VEL
LIN {X 0,Y 547.319,Z 711.46,A -85,B 0,C 180,E1 20859.389,E2 20859.389} C_VEL
LIN {X 0,Y 546.446,Z 704.659,A -85,B 0,C 180,E1 20859.229,E2 20859.229} C_VEL
LIN {X 0,Y 547.409,Z 658.896,A -85,B 0,C 180,E1 20855.705,E2 20855.705} C_VEL
LIN {X 0,Y 548.177,Z 621.777,A -85,B 0,C 180,E1 20852.828,E2 20852.828} C_VEL
LIN {X 0,Y 548.381,Z 588.082,A -85,B 0,C 180,E1 20850.329,E2 20850.329} C_VEL
LIN {X 0,Y 548.095,Z 553.969,A -85,B 0,C 180,E1 20847.961,E2 20847.961} C_VEL
LIN {X 0,Y 547.348,Z 527.315,A -85,B 0,C 180,E1 20846.219,E2 20846.219} C_VEL
LIN {X 0,Y 544.467,Z 515.687,A -85,B 0,C 180,E1 20845.396,E2 20845.396} C_VEL
LIN {X 0,Y 544.405,Z 515.238,A -85,B 0,C 180,E1 20845.168,E2 20845.168} C_VEL
LIN {X 0,Y 544.375,Z 515.234,A -85,B 0,C 180,E1 20841.824,E2 20841.824} C_VEL
LIN {X 0,Y 544.387,Z 515.23,A -85,B 0,C 180,E1 20838.377,E2 20838.377} C_VEL
LIN {X 0,Y 544.412,Z 515.441,A -85,B 0,C 180,E1 20835.148,E2 20835.148} C_VEL
LIN {X 0,Y 545.636,Z 518.614,A -85,B 0,C 180,E1 20834.685,E2 20834.685} C_VEL
LIN {X 0,Y 553.662,Z 536.184,A -85,B 0,C 180,E1 20832.387,E2 20832.387} C_VEL
LIN {X 0,Y 554.769,Z 538.926,A -85,B 0,C 180,E1 20832.052,E2 20832.052} C_VEL
LIN {X 0,Y 554.77,Z 544.072,A -85,B 0,C 180,E1 20831.673,E2 20831.673} C_VEL
LIN {X 0,Y 558.013,Z 559.248,A -85,B 0,C 180,E1 20831.117,E2 20831.117} C_VEL
LIN {X 0,Y 555.95,Z 767.492,A -85,B 0,C 180,E1 20827.883,E2 20827.883} C_VEL
LIN {X 0,Y 554.725,Z 892.219,A -85,B 0,C 180,E1 20825.966,E2 20825.966} C_VEL
LIN {X 0,Y 554.108,Z 915.745,A -85,B 0,C 180,E1 20825.416,E2 20825.416} C_VEL
LIN {X 0,Y 553.433,Z 937.717,A -85,B 0,C 180,E1 20824.716,E2 20824.716} C_VEL
LIN {X 0,Y 552.599,Z 958.769,A -85,B 0,C 180,E1 20823.85,E2 20823.85} C_VEL
LIN {X 0,Y 551.715,Z 978.559,A -85,B 0,C 180,E1 20822.873,E2 20822.873} C_VEL
LIN {X 0,Y 550.685,Z 1000.058,A -85,B 0,C 180,E1 20821.595,E2 20821.595} C_VEL
LIN {X 0,Y 549.669,Z 1020.187,A -85,B 0,C 180,E1 20820.196,E2 20820.196} C_VEL
LIN {X 0,Y 548.622,Z 1039.867,A -85,B 0,C 180,E1 20818.587,E2 20818.587} C_VEL
LIN {X 0,Y 547.595,Z 1059.199,A -85,B 0,C 180,E1 20816.765,E2 20816.765} C_VEL
LIN {X 0,Y 546.767,Z 1076.396,A -85,B 0,C 180,E1 20814.904,E2 20814.904} C_VEL
LIN {X 0,Y 545.989,Z 1092.365,A -85,B 0,C 180,E1 20812.909,E2 20812.909} C_VEL
LIN {X 0,Y 545.329,Z 1107.63,A -85,B 0,C 180,E1 20810.724,E2 20810.724} C_VEL
LIN {X 0,Y 544.857,Z 1120.367,A -85,B 0,C 180,E1 20808.621,E2 20808.621} C_VEL
LIN {X 0,Y 544.476,Z 1132.321,A -85,B 0,C 180,E1 20806.318,E2 20806.318} C_VEL
LIN {X 0,Y 544.23,Z 1142.337,A -85,B 0,C 180,E1 20804.062,E2 20804.062} C_VEL
LIN {X 0,Y 544.071,Z 1150.698,A -85,B 0,C 180,E1 20801.77,E2 20801.77} C_VEL
LIN {X 0,Y 543.962,Z 1157.474,A -85,B 0,C 180,E1 20799.522,E2 20799.522} C_VEL
LIN {X 0,Y 543.904,Z 1162.841,A -85,B 0,C 180,E1 20797.181,E2 20797.181} C_VEL
LIN {X 0,Y 543.914,Z 1166.436,A -85,B 0,C 180,E1 20795.062,E2 20795.062} C_VEL
LIN {X 0,Y 543.913,Z 1169.055,A -85,B 0,C 180,E1 20792.529,E2 20792.529} C_VEL
LIN {X 0,Y 543.892,Z 1169.939,A -85,B 0,C 180,E1 20790.316,E2 20790.316} C_VEL
LIN {X 0,Y 543.912,Z 1169.324,A -85,B 0,C 180,E1 20787.893,E2 20787.893} C_VEL
LIN {X 0,Y 543.913,Z 1167.389,A -85,B 0,C 180,E1 20785.678,E2 20785.678} C_VEL
LIN {X 0,Y 543.913,Z 1163.667,A -85,B 0,C 180,E1 20783.244,E2 20783.244} C_VEL
LIN {X 0,Y 543.968,Z 1159.062,A -85,B 0,C 180,E1 20781.118,E2 20781.118} C_VEL
LIN {X 0,Y 544.041,Z 1152.118,A -85,B 0,C 180,E1 20778.659,E2 20778.659} C_VEL
LIN {X 0,Y 544.169,Z 1144.52,A -85,B 0,C 180,E1 20776.506,E2 20776.506} C_VEL
LIN {X 0,Y 544.419,Z 1134.399,A -85,B 0,C 180,E1 20774.119,E2 20774.119} C_VEL
LIN {X 0,Y 544.747,Z 1123.984,A -85,B 0,C 180,E1 20772.04,E2 20772.04} C_VEL
LIN {X 0,Y 545.236,Z 1110.464,A -85,B 0,C 180,E1 20769.721,E2 20769.721} C_VEL
LIN {X 0,Y 545.839,Z 1096.217,A -85,B 0,C 180,E1 20767.604,E2 20767.604} C_VEL
LIN {X 0,Y 546.55,Z 1080.408,A -85,B 0,C 180,E1 20765.578,E2 20765.578} C_VEL
LIN {X 0,Y 547.46,Z 1062.116,A -85,B 0,C 180,E1 20763.536,E2 20763.536} C_VEL
LIN {X 0,Y 548.429,Z 1043.897,A -85,B 0,C 180,E1 20761.764,E2 20761.764} C_VEL
LIN {X 0,Y 549.413,Z 1024.598,A -85,B 0,C 180,E1 20760.15,E2 20760.15} C_VEL
LIN {X 0,Y 550.536,Z 1003.11,A -85,B 0,C 180,E1 20758.604,E2 20758.604} C_VEL
LIN {X 0,Y 551.474,Z 983.818,A -85,B 0,C 180,E1 20757.42,E2 20757.42} C_VEL
LIN {X 0,Y 552.439,Z 962.236,A -85,B 0,C 180,E1 20756.307,E2 20756.307} C_VEL
LIN {X 0,Y 553.254,Z 942.442,A -85,B 0,C 180,E1 20755.466,E2 20755.466} C_VEL
LIN {X 0,Y 554.01,Z 918.697,A -85,B 0,C 180,E1 20754.666,E2 20754.666} C_VEL
LIN {X 0,Y 554.634,Z 896.615,A -85,B 0,C 180,E1 20754.118,E2 20754.118} C_VEL
LIN {X 0,Y 555.082,Z 861.188,A -85,B 0,C 180,E1 20753.538,E2 20753.538} C_VEL
LIN {X 0,Y 557.084,Z 651.18,A -85,B 0,C 180,E1 20750.325,E2 20750.325} C_VEL
LIN {X 0,Y 557.912,Z 555.131,A -85,B 0,C 180,E1 20748.805,E2 20748.805} C_VEL
LIN {X 0,Y 555.565,Z 542.265,A -85,B 0,C 180,E1 20748.364,E2 20748.364} C_VEL
LIN {X 0,Y 555.479,Z 538.548,A -85,B 0,C 180,E1 20748.102,E2 20748.102} C_VEL
LIN {X 0,Y 547.557,Z 522.476,A -85,B 0,C 180,E1 20746.206,E2 20746.206} C_VEL
LIN {X 0,Y 544.454,Z 515.615,A -85,B 0,C 180,E1 20745.373,E2 20745.373} C_VEL
LIN {X 0,Y 544.381,Z 515.213,A -85,B 0,C 180,E1 20744.849,E2 20744.849} C_VEL
LIN {X 0,Y 544.398,Z 515.222,A -85,B 0,C 180,E1 20741.466,E2 20741.466} C_VEL
LIN {X 0,Y 544.399,Z 515.227,A -85,B 0,C 180,E1 20737.971,E2 20737.971} C_VEL
LIN {X 0,Y 544.388,Z 515.234,A -85,B 0,C 180,E1 20734.578,E2 20734.578} C_VEL
LIN {X 0,Y 544.388,Z 515.23,A -85,B 0,C 180,E1 20731.317,E2 20731.317} C_VEL
LIN {X 0,Y 544.384,Z 515.227,A -85,B 0,C 180,E1 20728.046,E2 20728.046} C_VEL
LIN {X 0,Y 544.389,Z 515.234,A -85,B 0,C 180,E1 20724.756,E2 20724.756} C_VEL
LIN {X 0,Y 544.395,Z 515.218,A -85,B 0,C 180,E1 20721.324,E2 20721.324} C_VEL
LIN {X 0,Y 544.397,Z 515.23,A -85,B 0,C 180,E1 20717.861,E2 20717.861} C_VEL
LIN {X 0,Y 544.384,Z 515.224,A -85,B 0,C 180,E1 20714.465,E2 20714.465} C_VEL
LIN {X 0,Y 544.388,Z 515.233,A -85,B 0,C 180,E1 20711.119,E2 20711.119} C_VEL
LIN {X 0,Y 544.386,Z 515.222,A -85,B 0,C 180,E1 20707.811,E2 20707.811} C_VEL
LIN {X 0,Y 544.397,Z 515.238,A -85,B 0,C 180,E1 20704.424,E2 20704.424} C_VEL
LIN {X 0,Y 544.399,Z 515.23,A -85,B 0,C 180,E1 20700.947,E2 20700.947} C_VEL
LIN {X 0,Y 544.385,Z 515.234,A -85,B 0,C 180,E1 20697.579,E2 20697.579} C_VEL
LIN {X 0,Y 544.389,Z 515.234,A -85,B 0,C 180,E1 20694.202,E2 20694.202} C_VEL
LIN {X 0,Y 544.383,Z 515.233,A -85,B 0,C 180,E1 20690.912,E2 20690.912} C_VEL
LIN {X 0,Y 544.398,Z 515.216,A -85,B 0,C 180,E1 20687.483,E2 20687.483} C_VEL
LIN {X 0,Y 544.401,Z 515.23,A -85,B 0,C 180,E1 20684.008,E2 20684.008} C_VEL
LIN {X 0,Y 544.378,Z 515.219,A -85,B 0,C 180,E1 20680.583,E2 20680.583} C_VEL
LIN {X 0,Y 544.392,Z 515.234,A -85,B 0,C 180,E1 20677.313,E2 20677.313} C_VEL
LIN {X 0,Y 544.381,Z 515.224,A -85,B 0,C 180,E1 20673.962,E2 20673.962} C_VEL
LIN {X 0,Y 544.401,Z 515.228,A -85,B 0,C 180,E1 20670.514,E2 20670.514} C_VEL
LIN {X 0,Y 544.396,Z 515.217,A -85,B 0,C 180,E1 20669.079,E2 20669.079} C_VEL
LIN {X 0,Y 543.38,Z 515.35,A -85,B 0,C 180,E1 20668.268,E2 20668.268} C_VEL
LIN {X 0,Y 536.952,Z 516.162,A -85,B 0,C 180,E1 20665.991,E2 20665.991} C_VEL
LIN {X 0,Y 536.445,Z 516.217,A -85,B 0,C 180,E1 20665.398,E2 20665.398} C_VEL
LIN {X 0,Y 536.452,Z 516.226,A -85,B 0,C 180,E1 20661.864,E2 20661.864} C_VEL
LIN {X 0,Y 536.458,Z 516.22,A -85,B 0,C 180,E1 20658.431,E2 20658.431} C_VEL
LIN {X 0,Y 536.435,Z 516.216,A -85,B 0,C 180,E1 20655.056,E2 20655.056} C_VEL
LIN {X 0,Y 536.464,Z 516.418,A -85,B 0,C 180,E1 20653.062,E2 20653.062} C_VEL
LIN {X 0,Y 537.796,Z 519.75,A -85,B 0,C 180,E1 20652.588,E2 20652.588} C_VEL
LIN {X 0,Y 545.278,Z 535.576,A -85,B 0,C 180,E1 20650.611,E2 20650.611} C_VEL
LIN {X 0,Y 547.596,Z 541.126,A -85,B 0,C 180,E1 20649.973,E2 20649.973} C_VEL
LIN {X 0,Y 545.825,Z 587.321,A -85,B 0,C 180,E1 20646.734,E2 20646.734} C_VEL
LIN {X 0,Y 545.944,Z 591.05,A -85,B 0,C 180,E1 20646.528,E2 20646.528} C_VEL
LIN {X 0,Y 548.137,Z 604.443,A -85,B 0,C 180,E1 20646.145,E2 20646.145} C_VEL
LIN {X 0,Y 545.946,Z 835.724,A -85,B 0,C 180,E1 20642.694,E2 20642.694} C_VEL
LIN {X 0,Y 545.331,Z 897.281,A -85,B 0,C 180,E1 20641.758,E2 20641.758} C_VEL
LIN {X 0,Y 544.734,Z 918.903,A -85,B 0,C 180,E1 20641.232,E2 20641.232} C_VEL
LIN {X 0,Y 544.056,Z 940.369,A -85,B 0,C 180,E1 20640.51,E2 20640.51} C_VEL
LIN {X 0,Y 543.282,Z 959.966,A -85,B 0,C 180,E1 20639.674,E2 20639.674} C_VEL
LIN {X 0,Y 542.397,Z 979.506,A -85,B 0,C 180,E1 20638.639,E2 20638.639} C_VEL
LIN {X 0,Y 541.397,Z 999.957,A -85,B 0,C 180,E1 20637.337,E2 20637.337} C_VEL
LIN {X 0,Y 540.491,Z 1018.173,A -85,B 0,C 180,E1 20635.966,E2 20635.966} C_VEL
LIN {X 0,Y 539.526,Z 1036.41,A -85,B 0,C 180,E1 20634.345,E2 20634.345} C_VEL
LIN {X 0,Y 538.652,Z 1053.28,A -85,B 0,C 180,E1 20632.597,E2 20632.597} C_VEL
LIN {X 0,Y 537.885,Z 1069.186,A -85,B 0,C 180,E1 20630.682,E2 20630.682} C_VEL
LIN {X 0,Y 537.278,Z 1083.384,A -85,B 0,C 180,E1 20628.695,E2 20628.695} C_VEL
LIN {X 0,Y 536.799,Z 1095.704,A -85,B 0,C 180,E1 20626.669,E2 20626.669} C_VEL
LIN {X 0,Y 536.428,Z 1107.105,A -85,B 0,C 180,E1 20624.464,E2 20624.464} C_VEL
LIN {X 0,Y 536.184,Z 1116.587,A -85,B 0,C 180,E1 20622.274,E2 20622.274} C_VEL
LIN {X 0,Y 536.039,Z 1124.236,A -85,B 0,C 180,E1 20620.098,E2 20620.098} C_VEL
LIN {X 0,Y 535.959,Z 1130.54,A -85,B 0,C 180,E1 20617.827,E2 20617.827} C_VEL
LIN {X 0,Y 535.922,Z 1135.249,A -85,B 0,C 180,E1 20615.567,E2 20615.567} C_VEL
LIN {X 0,Y 535.911,Z 1138.238,A -85,B 0,C 180,E1 20613.316,E2 20613.316} C_VEL
LIN {X 0,Y 535.907,Z 1139.794,A -85,B 0,C 180,E1 20610.962,E2 20610.962} C_VEL
LIN {X 0,Y 535.908,Z 1139.747,A -85,B 0,C 180,E1 20608.717,E2 20608.717} C_VEL
LIN {X 0,Y 535.91,Z 1138.109,A -85,B 0,C 180,E1 20606.47,E2 20606.47} C_VEL
LIN {X 0,Y 535.928,Z 1135.014,A -85,B 0,C 180,E1 20604.218,E2 20604.218} C_VEL
LIN {X 0,Y 535.969,Z 1130.242,A -85,B 0,C 180,E1 20601.957,E2 20601.957} C_VEL
LIN {X 0,Y 536.054,Z 1123.469,A -85,B 0,C 180,E1 20599.576,E2 20599.576} C_VEL
LIN {X 0,Y 536.212,Z 1115.667,A -85,B 0,C 180,E1 20597.399,E2 20597.399} C_VEL
LIN {X 0,Y 536.461,Z 1105.97,A -85,B 0,C 180,E1 20595.206,E2 20595.206} C_VEL
LIN {X 0,Y 536.84,Z 1094.312,A -85,B 0,C 180,E1 20592.998,E2 20592.998} C_VEL
LIN {X 0,Y 537.364,Z 1081.137,A -85,B 0,C 180,E1 20590.884,E2 20590.884} C_VEL
LIN {X 0,Y 538.026,Z 1066.642,A -85,B 0,C 180,E1 20588.893,E2 20588.893} C_VEL
LIN {X 0,Y 538.772,Z 1051.031,A -85,B 0,C 180,E1 20587.063,E2 20587.063} C_VEL
LIN {X 0,Y 539.654,Z 1033.64,A -85,B 0,C 180,E1 20585.304,E2 20585.304} C_VEL
LIN {X 0,Y 540.64,Z 1015.04,A -85,B 0,C 180,E1 20583.697,E2 20583.697} C_VEL
LIN {X 0,Y 541.578,Z 996.807,A -85,B 0,C 180,E1 20582.351,E2 20582.351} C_VEL
LIN {X 0,Y 542.508,Z 976.989,A -85,B 0,C 180,E1 20581.127,E2 20581.127} C_VEL
LIN {X 0,Y 543.465,Z 955.49,A -85,B 0,C 180,E1 20580.033,E2 20580.033} C_VEL
LIN {X 0,Y 544.274,Z 934.727,A -85,B 0,C 180,E1 20579.186,E2 20579.186} C_VEL
LIN {X 0,Y 544.902,Z 913.692,A -85,B 0,C 180,E1 20578.535,E2 20578.535} C_VEL
LIN {X 0,Y 545.402,Z 891.425,A -85,B 0,C 180,E1 20578.05,E2 20578.05} C_VEL
LIN {X 0,Y 547.454,Z 672.421,A -85,B 0,C 180,E1 20574.788,E2 20574.788} C_VEL
LIN {X 0,Y 547.92,Z 604.823,A -85,B 0,C 180,E1 20573.754,E2 20573.754} C_VEL
LIN {X 0,Y 544.919,Z 590.53,A -85,B 0,C 180,E1 20573.261,E2 20573.261} C_VEL
LIN {X 0,Y 546.539,Z 550.461,A -85,B 0,C 180,E1 20569.881,E2 20569.881} C_VEL
LIN {X 0,Y 546.856,Z 540.883,A -85,B 0,C 180,E1 20569.036,E2 20569.036} C_VEL
LIN {X 0,Y 539.594,Z 523.787,A -85,B 0,C 180,E1 20566.717,E2 20566.717} C_VEL
LIN {X 0,Y 536.499,Z 516.579,A -85,B 0,C 180,E1 20565.663,E2 20565.663} C_VEL
LIN {X 0,Y 536.423,Z 516.23,A -85,B 0,C 180,E1 20564.795,E2 20564.795} C_VEL
LIN {X 0,Y 536.422,Z 516.189,A -85,B 0,C 180,E1 20561.631,E2 20561.631} C_VEL
LIN {X 0,Y 536.403,Z 516.223,A -85,B 0,C 180,E1 20558.232,E2 20558.232} C_VEL
LIN {X 0,Y 536.437,Z 516.475,A -85,B 0,C 180,E1 20556.134,E2 20556.134} C_VEL
LIN {X 0,Y 542.181,Z 534.112,A -85,B 0,C 180,E1 20554.354,E2 20554.354} C_VEL
LIN {X 0,Y 541.702,Z 572.289,A -85,B 0,C 180,E1 20551.367,E2 20551.367} C_VEL
LIN {X 0,Y 540.984,Z 613.78,A -85,B 0,C 180,E1 20548.119,E2 20548.119} C_VEL
LIN {X 0,Y 540.04,Z 654.986,A -85,B 0,C 180,E1 20544.876,E2 20544.876} C_VEL
LIN {X 0,Y 538.986,Z 698.835,A -85,B 0,C 180,E1 20541.435,E2 20541.435} C_VEL
LIN {X 0,Y 538.891,Z 705.732,A -85,B 0,C 180,E1 20540.938,E2 20540.938} C_VEL
LIN {X 0,Y 539.987,Z 715.611,A -85,B 0,C 180,E1 20540.756,E2 20540.756} C_VEL
LIN {X 0,Y 539.155,Z 875.994,A -85,B 0,C 180,E1 20538.536,E2 20538.536} C_VEL
LIN {X 0,Y 538.886,Z 893.107,A -85,B 0,C 180,E1 20538.1,E2 20538.1} C_VEL
LIN {X 0,Y 538.515,Z 910.584,A -85,B 0,C 180,E1 20537.449,E2 20537.449} C_VEL
LIN {X 0,Y 538.108,Z 926.812,A -85,B 0,C 180,E1 20536.628,E2 20536.628} C_VEL
LIN {X 0,Y 537.638,Z 942.74,A -85,B 0,C 180,E1 20535.589,E2 20535.589} C_VEL
LIN {X 0,Y 537.198,Z 957.987,A -85,B 0,C 180,E1 20534.333,E2 20534.333} C_VEL
LIN {X 0,Y 536.815,Z 970.826,A -85,B 0,C 180,E1 20533.025,E2 20533.025} C_VEL
LIN {X 0,Y 536.499,Z 982.22,A -85,B 0,C 180,E1 20531.612,E2 20531.612} C_VEL
LIN {X 0,Y 536.25,Z 992.884,A -85,B 0,C 180,E1 20529.986,E2 20529.986} C_VEL
LIN {X 0,Y 536.074,Z 1001.875,A -85,B 0,C 180,E1 20528.257,E2 20528.257} C_VEL
LIN {X 0,Y 535.977,Z 1008.816,A -85,B 0,C 180,E1 20526.534,E2 20526.534} C_VEL
LIN {X 0,Y 535.93,Z 1014.232,A -85,B 0,C 180,E1 20524.709,E2 20524.709} C_VEL
LIN {X 0,Y 535.916,Z 1017.974,A -85,B 0,C 180,E1 20522.781,E2 20522.781} C_VEL
LIN {X 0,Y 535.914,Z 1019.78,A -85,B 0,C 180,E1 20520.855,E2 20520.855} C_VEL
LIN {X 0,Y 535.916,Z 1019.732,A -85,B 0,C 180,E1 20519.038,E2 20519.038} C_VEL
LIN {X 0,Y 535.916,Z 1018.107,A -85,B 0,C 180,E1 20517.22,E2 20517.22} C_VEL
LIN {X 0,Y 535.93,Z 1014.451,A -85,B 0,C 180,E1 20515.292,E2 20515.292} C_VEL
LIN {X 0,Y 535.97,Z 1009.448,A -85,B 0,C 180,E1 20513.574,E2 20513.574} C_VEL
LIN {X 0,Y 536.062,Z 1002.785,A -85,B 0,C 180,E1 20511.851,E2 20511.851} C_VEL
LIN {X 0,Y 536.226,Z 994.037,A -85,B 0,C 180,E1 20510.123,E2 20510.123} C_VEL
LIN {X 0,Y 536.463,Z 983.641,A -85,B 0,C 180,E1 20508.497,E2 20508.497} C_VEL
LIN {X 0,Y 536.792,Z 971.358,A -85,B 0,C 180,E1 20506.95,E2 20506.95} C_VEL
LIN {X 0,Y 537.122,Z 960.007,A -85,B 0,C 180,E1 20505.776,E2 20505.776} C_VEL
LIN {X 0,Y 537.48,Z 948.087,A -85,B 0,C 180,E1 20504.739,E2 20504.739} C_VEL
LIN {X 0,Y 537.905,Z 933.695,A -85,B 0,C 180,E1 20503.7,E2 20503.7} C_VEL
LIN {X 0,Y 538.312,Z 918.153,A -85,B 0,C 180,E1 20502.823,E2 20502.823} C_VEL
LIN {X 0,Y 538.678,Z 903.358,A -85,B 0,C 180,E1 20502.166,E2 20502.166} C_VEL
LIN {X 0,Y 539.018,Z 885.2,A -85,B 0,C 180,E1 20501.586,E2 20501.586} C_VEL
LIN {X 0,Y 539.215,Z 868.439,A -85,B 0,C 180,E1 20501.246,E2 20501.246} C_VEL
LIN {X 0,Y 539.825,Z 712.394,A -85,B 0,C 180,E1 20499.103,E2 20499.103} C_VEL
LIN {X 0,Y 538.828,Z 704.754,A -85,B 0,C 180,E1 20498.929,E2 20498.929} C_VEL
LIN {X 0,Y 539.942,Z 659.727,A -85,B 0,C 180,E1 20495.4,E2 20495.4} C_VEL
LIN {X 0,Y 540.629,Z 622.385,A -85,B 0,C 180,E1 20492.533,E2 20492.533} C_VEL
LIN {X 0,Y 540.755,Z 588.498,A -85,B 0,C 180,E1 20490.051,E2 20490.051} C_VEL
LIN {X 0,Y 540.405,Z 552.075,A -85,B 0,C 180,E1 20487.551,E2 20487.551} C_VEL
LIN {X 0,Y 539.697,Z 529.501,A -85,B 0,C 180,E1 20486.097,E2 20486.097} C_VEL
LIN {X 0,Y 536.543,Z 516.719,A -85,B 0,C 180,E1 20485.201,E2 20485.201} C_VEL
LIN {X 0,Y 536.455,Z 516.228,A -85,B 0,C 180,E1 20484.967,E2 20484.967} C_VEL
LIN {X 0,Y 536.45,Z 516.214,A -85,B 0,C 180,E1 20481.636,E2 20481.636} C_VEL
LIN {X 0,Y 536.443,Z 516.221,A -85,B 0,C 180,E1 20478.206,E2 20478.206} C_VEL
LIN {X 0,Y 536.49,Z 516.458,A -85,B 0,C 180,E1 20475.875,E2 20475.875} C_VEL
LIN {X 0,Y 537.906,Z 519.914,A -85,B 0,C 180,E1 20475.363,E2 20475.363} C_VEL
LIN {X 0,Y 547.091,Z 539.976,A -85,B 0,C 180,E1 20472.691,E2 20472.691} C_VEL
LIN {X 0,Y 548.183,Z 542.899,A -85,B 0,C 180,E1 20472.338,E2 20472.338} C_VEL
LIN {X 0,Y 551.962,Z 561.153,A -85,B 0,C 180,E1 20471.635,E2 20471.635} C_VEL
LIN {X 0,Y 549.614,Z 769.525,A -85,B 0,C 180,E1 20468.365,E2 20468.365} C_VEL
LIN {X 0,Y 548.242,Z 892.314,A -85,B 0,C 180,E1 20466.458,E2 20466.458} C_VEL
LIN {X 0,Y 547.56,Z 915.743,A -85,B 0,C 180,E1 20465.905,E2 20465.905} C_VEL
LIN {X 0,Y 546.782,Z 937.72,A -85,B 0,C 180,E1 20465.2,E2 20465.2} C_VEL
LIN {X 0,Y 545.868,Z 958.391,A -85,B 0,C 180,E1 20464.344,E2 20464.344} C_VEL
LIN {X 0,Y 544.921,Z 977.444,A -85,B 0,C 180,E1 20463.399,E2 20463.399} C_VEL
LIN {X 0,Y 543.719,Z 999.244,A -85,B 0,C 180,E1 20462.104,E2 20462.104} C_VEL
LIN {X 0,Y 542.586,Z 1019.403,A -85,B 0,C 180,E1 20460.694,E2 20460.694} C_VEL
LIN {X 0,Y 541.366,Z 1039.27,A -85,B 0,C 180,E1 20459.061,E2 20459.061} C_VEL
LIN {X 0,Y 540.2,Z 1058.79,A -85,B 0,C 180,E1 20457.205,E2 20457.205} C_VEL
LIN {X 0,Y 539.251,Z 1075.66,A -85,B 0,C 180,E1 20455.361,E2 20455.361} C_VEL
LIN {X 0,Y 538.34,Z 1091.994,A -85,B 0,C 180,E1 20453.304,E2 20453.304} C_VEL
LIN {X 0,Y 537.604,Z 1106.923,A -85,B 0,C 180,E1 20451.15,E2 20451.15} C_VEL
LIN {X 0,Y 537.052,Z 1119.73,A -85,B 0,C 180,E1 20449.015,E2 20449.015} C_VEL
LIN {X 0,Y 536.601,Z 1131.801,A -85,B 0,C 180,E1 20446.676,E2 20446.676} C_VEL
LIN {X 0,Y 536.312,Z 1141.533,A -85,B 0,C 180,E1 20444.467,E2 20444.467} C_VEL
LIN {X 0,Y 536.096,Z 1150.343,A -85,B 0,C 180,E1 20442.057,E2 20442.057} C_VEL
LIN {X 0,Y 535.976,Z 1156.868,A -85,B 0,C 180,E1 20439.882,E2 20439.882} C_VEL
LIN {X 0,Y 535.917,Z 1162.634,A -85,B 0,C 180,E1 20437.396,E2 20437.396} C_VEL
LIN {X 0,Y 535.914,Z 1166.277,A -85,B 0,C 180,E1 20435.245,E2 20435.245} C_VEL
LIN {X 0,Y 535.898,Z 1168.92,A -85,B 0,C 180,E1 20432.781,E2 20432.781} C_VEL
LIN {X 0,Y 535.884,Z 1169.872,A -85,B 0,C 180,E1 20430.641,E2 20430.641} C_VEL
LIN {X 0,Y 535.905,Z 1169.526,A -85,B 0,C 180,E1 20428.182,E2 20428.182} C_VEL
LIN {X 0,Y 535.917,Z 1167.616,A -85,B 0,C 180,E1 20425.827,E2 20425.827} C_VEL
LIN {X 0,Y 535.922,Z 1164.08,A -85,B 0,C 180,E1 20423.358,E2 20423.358} C_VEL
LIN {X 0,Y 535.972,Z 1159.572,A -85,B 0,C 180,E1 20421.201,E2 20421.201} C_VEL
LIN {X 0,Y 536.051,Z 1153.177,A -85,B 0,C 180,E1 20418.815,E2 20418.815} C_VEL
LIN {X 0,Y 536.197,Z 1145.339,A -85,B 0,C 180,E1 20416.521,E2 20416.521} C_VEL
LIN {X 0,Y 536.469,Z 1135.942,A -85,B 0,C 180,E1 20414.21,E2 20414.21} C_VEL
LIN {X 0,Y 536.841,Z 1125.147,A -85,B 0,C 180,E1 20411.991,E2 20411.991} C_VEL
LIN {X 0,Y 537.393,Z 1111.864,A -85,B 0,C 180,E1 20409.639,E2 20409.639} C_VEL
LIN {X 0,Y 538.012,Z 1098.56,A -85,B 0,C 180,E1 20407.606,E2 20407.606} C_VEL
LIN {X 0,Y 538.864,Z 1082.266,A -85,B 0,C 180,E1 20405.441,E2 20405.441} C_VEL
LIN {X 0,Y 539.84,Z 1065.434,A -85,B 0,C 180,E1 20403.489,E2 20403.489} C_VEL
LIN {X 0,Y 540.864,Z 1047.575,A -85,B 0,C 180,E1 20401.694,E2 20401.694} C_VEL
LIN {X 0,Y 542.075,Z 1027.526,A -85,B 0,C 180,E1 20399.948,E2 20399.948} C_VEL
LIN {X 0,Y 543.281,Z 1007.477,A -85,B 0,C 180,E1 20398.441,E2 20398.441} C_VEL
LIN {X 0,Y 544.416,Z 986.83,A -85,B 0,C 180,E1 20397.132,E2 20397.132} C_VEL
LIN {X 0,Y 545.495,Z 966.056,A -85,B 0,C 180,E1 20396.01,E2 20396.01} C_VEL
LIN {X 0,Y 546.458,Z 945.196,A -85,B 0,C 180,E1 20395.093,E2 20395.093} C_VEL
LIN {X 0,Y 547.351,Z 922.896,A -85,B 0,C 180,E1 20394.301,E2 20394.301} C_VEL
LIN {X 0,Y 547.981,Z 900.836,A -85,B 0,C 180,E1 20393.719,E2 20393.719} C_VEL
LIN {X 0,Y 548.531,Z 872.893,A -85,B 0,C 180,E1 20393.219,E2 20393.219} C_VEL
LIN {X 0,Y 550.816,Z 660.915,A -85,B 0,C 180,E1 20389.944,E2 20389.944} C_VEL
LIN {X 0,Y 551.871,Z 556.85,A -85,B 0,C 180,E1 20388.283,E2 20388.283} C_VEL
LIN {X 0,Y 549.075,Z 542.529,A -85,B 0,C 180,E1 20387.77,E2 20387.77} C_VEL
LIN {X 0,Y 539.969,Z 524.039,A -85,B 0,C 180,E1 20385.577,E2 20385.577} C_VEL
LIN {X 0,Y 537.88,Z 519.882,A -85,B 0,C 180,E1 20385.059,E2 20385.059} C_VEL
LIN {X 0,Y 536.486,Z 516.45,A -85,B 0,C 180,E1 20384.607,E2 20384.607} C_VEL
LIN {X 0,Y 536.464,Z 516.206,A -85,B 0,C 180,E1 20381.283,E2 20381.283} C_VEL
LIN {X 0,Y 536.453,Z 516.212,A -85,B 0,C 180,E1 20377.789,E2 20377.789} C_VEL
LIN {X 0,Y 536.446,Z 516.226,A -85,B 0,C 180,E1 20374.384,E2 20374.384} C_VEL
LIN {X 0,Y 536.454,Z 516.22,A -85,B 0,C 180,E1 20370.978,E2 20370.978} C_VEL
LIN {X 0,Y 536.46,Z 516.206,A -85,B 0,C 180,E1 20367.479,E2 20367.479} C_VEL
LIN {X 0,Y 536.452,Z 516.222,A -85,B 0,C 180,E1 20364.037,E2 20364.037} C_VEL
LIN {X 0,Y 536.448,Z 516.213,A -85,B 0,C 180,E1 20360.665,E2 20360.665} C_VEL
LIN {X 0,Y 536.453,Z 516.221,A -85,B 0,C 180,E1 20357.238,E2 20357.238} C_VEL
LIN {X 0,Y 536.463,Z 516.211,A -85,B 0,C 180,E1 20353.802,E2 20353.802} C_VEL
LIN {X 0,Y 536.449,Z 516.212,A -85,B 0,C 180,E1 20350.307,E2 20350.307} C_VEL
LIN {X 0,Y 536.448,Z 516.211,A -85,B 0,C 180,E1 20346.958,E2 20346.958} C_VEL
LIN {X 0,Y 536.445,Z 516.217,A -85,B 0,C 180,E1 20343.633,E2 20343.633} C_VEL
LIN {X 0,Y 536.461,Z 516.223,A -85,B 0,C 180,E1 20340.213,E2 20340.213} C_VEL
LIN {X 0,Y 536.459,Z 516.217,A -85,B 0,C 180,E1 20336.687,E2 20336.687} C_VEL
LIN {X 0,Y 536.444,Z 516.218,A -85,B 0,C 180,E1 20333.256,E2 20333.256} C_VEL
LIN {X 0,Y 536.453,Z 516.224,A -85,B 0,C 180,E1 20329.909,E2 20329.909} C_VEL
LIN {X 0,Y 536.448,Z 516.209,A -85,B 0,C 180,E1 20326.527,E2 20326.527} C_VEL
LIN {X 0,Y 536.458,Z 516.221,A -85,B 0,C 180,E1 20323.097,E2 20323.097} C_VEL
LIN {X 0,Y 536.457,Z 516.207,A -85,B 0,C 180,E1 20319.637,E2 20319.637} C_VEL
LIN {X 0,Y 536.44,Z 516.217,A -85,B 0,C 180,E1 20316.376,E2 20316.376} C_VEL
LIN {X 0,Y 536.456,Z 516.216,A -85,B 0,C 180,E1 20312.949,E2 20312.949} C_VEL
LIN {X 0,Y 536.442,Z 516.207,A -85,B 0,C 180,E1 20309.652,E2 20309.652} C_VEL
LIN {X 0,Y 536.459,Z 516.225,A -85,B 0,C 180,E1 20306.229,E2 20306.229} C_VEL
LIN {X 0,Y 536.445,Z 516.217,A -85,B 0,C 180,E1 20305.398,E2 20305.398} C_VEL
LIN {X 0,Y 535.49,Z 516.337,A -85,B 0,C 180,E1 20304.575,E2 20304.575} C_VEL
LIN {X 0,Y 528.96,Z 517.161,A -85,B 0,C 180,E1 20302.204,E2 20302.204} C_VEL
LIN {X 0,Y 528.503,Z 517.214,A -85,B 0,C 180,E1 20301.662,E2 20301.662} C_VEL
LIN {X 0,Y 528.518,Z 517.211,A -85,B 0,C 180,E1 20298.247,E2 20298.247} C_VEL
LIN {X 0,Y 528.505,Z 517.206,A -85,B 0,C 180,E1 20294.81,E2 20294.81} C_VEL
LIN {X 0,Y 528.572,Z 517.547,A -85,B 0,C 180,E1 20293.775,E2 20293.775} C_VEL
LIN {X 0,Y 530.108,Z 521.117,A -85,B 0,C 180,E1 20293.277,E2 20293.277} C_VEL
LIN {X 0,Y 537.962,Z 537.719,A -85,B 0,C 180,E1 20291.144,E2 20291.144} C_VEL
LIN {X 0,Y 541.005,Z 544.763,A -85,B 0,C 180,E1 20290.305,E2 20290.305} C_VEL
LIN {X 0,Y 539.062,Z 589.234,A -85,B 0,C 180,E1 20287.138,E2 20287.138} C_VEL
LIN {X 0,Y 541.665,Z 605.922,A -85,B 0,C 180,E1 20286.623,E2 20286.623} C_VEL
LIN {X 0,Y 539.202,Z 837.301,A -85,B 0,C 180,E1 20283.132,E2 20283.132} C_VEL
LIN {X 0,Y 538.528,Z 897.316,A -85,B 0,C 180,E1 20282.207,E2 20282.207} C_VEL
LIN {X 0,Y 537.861,Z 919.072,A -85,B 0,C 180,E1 20281.673,E2 20281.673} C_VEL
LIN {X 0,Y 537.112,Z 940.385,A -85,B 0,C 180,E1 20280.948,E2 20280.948} C_VEL
LIN {X 0,Y 536.249,Z 960.055,A -85,B 0,C 180,E1 20280.1,E2 20280.1} C_VEL
LIN {X 0,Y 535.241,Z 979.753,A -85,B 0,C 180,E1 20279.044,E2 20279.044} C_VEL
LIN {X 0,Y 534.119,Z 1000.221,A -85,B 0,C 180,E1 20277.722,E2 20277.722} C_VEL
LIN {X 0,Y 533.057,Z 1019.099,A -85,B 0,C 180,E1 20276.274,E2 20276.274} C_VEL
LIN {X 0,Y 532,Z 1036.947,A -85,B 0,C 180,E1 20274.66,E2 20274.66} C_VEL
LIN {X 0,Y 531.042,Z 1053.286,A -85,B 0,C 180,E1 20272.939,E2 20272.939} C_VEL
LIN {X 0,Y 530.176,Z 1069.192,A -85,B 0,C 180,E1 20270.997,E2 20270.997} C_VEL
LIN {X 0,Y 529.506,Z 1082.836,A -85,B 0,C 180,E1 20269.067,E2 20269.067} C_VEL
LIN {X 0,Y 528.934,Z 1095.507,A -85,B 0,C 180,E1 20266.96,E2 20266.96} C_VEL
LIN {X 0,Y 528.505,Z 1107.109,A -85,B 0,C 180,E1 20264.685,E2 20264.685} C_VEL
LIN {X 0,Y 528.23,Z 1116.59,A -85,B 0,C 180,E1 20262.462,E2 20262.462} C_VEL
LIN {X 0,Y 528.064,Z 1124.238,A -85,B 0,C 180,E1 20260.252,E2 20260.252} C_VEL
LIN {X 0,Y 527.968,Z 1130.594,A -85,B 0,C 180,E1 20257.924,E2 20257.924} C_VEL
LIN {X 0,Y 527.926,Z 1135.25,A -85,B 0,C 180,E1 20255.652,E2 20255.652} C_VEL
LIN {X 0,Y 527.91,Z 1138.239,A -85,B 0,C 180,E1 20253.366,E2 20253.366} C_VEL
LIN {X 0,Y 527.908,Z 1139.794,A -85,B 0,C 180,E1 20250.977,E2 20250.977} C_VEL
LIN {X 0,Y 527.908,Z 1139.746,A -85,B 0,C 180,E1 20248.698,E2 20248.698} C_VEL
LIN {X 0,Y 527.909,Z 1138.108,A -85,B 0,C 180,E1 20246.417,E2 20246.417} C_VEL
LIN {X 0,Y 527.929,Z 1135.013,A -85,B 0,C 180,E1 20244.13,E2 20244.13} C_VEL
LIN {X 0,Y 527.975,Z 1130.241,A -85,B 0,C 180,E1 20241.834,E2 20241.834} C_VEL
LIN {X 0,Y 528.078,Z 1123.466,A -85,B 0,C 180,E1 20239.417,E2 20239.417} C_VEL
LIN {X 0,Y 528.26,Z 1115.664,A -85,B 0,C 180,E1 20237.206,E2 20237.206} C_VEL
LIN {X 0,Y 528.542,Z 1105.968,A -85,B 0,C 180,E1 20234.979,E2 20234.979} C_VEL
LIN {X 0,Y 528.977,Z 1094.306,A -85,B 0,C 180,E1 20232.737,E2 20232.737} C_VEL
LIN {X 0,Y 529.545,Z 1081.902,A -85,B 0,C 180,E1 20230.705,E2 20230.705} C_VEL
LIN {X 0,Y 530.24,Z 1068.149,A -85,B 0,C 180,E1 20228.774,E2 20228.774} C_VEL
LIN {X 0,Y 531.089,Z 1052.512,A -85,B 0,C 180,E1 20226.883,E2 20226.883} C_VEL
LIN {X 0,Y 532.105,Z 1034.849,A -85,B 0,C 180,E1 20225.048,E2 20225.048} C_VEL
LIN {X 0,Y 533.195,Z 1016.743,A -85,B 0,C 180,E1 20223.442,E2 20223.442} C_VEL
LIN {X 0,Y 534.241,Z 998.315,A -85,B 0,C 180,E1 20222.052,E2 20222.052} C_VEL
LIN {X 0,Y 535.281,Z 978.986,A -85,B 0,C 180,E1 20220.822,E2 20220.822} C_VEL
LIN {X 0,Y 536.282,Z 959.303,A -85,B 0,C 180,E1 20219.775,E2 20219.775} C_VEL
LIN {X 0,Y 537.158,Z 939.418,A -85,B 0,C 180,E1 20218.925,E2 20218.925} C_VEL
LIN {X 0,Y 537.92,Z 917.302,A -85,B 0,C 180,E1 20218.188,E2 20218.188} C_VEL
LIN {X 0,Y 538.556,Z 895.699,A -85,B 0,C 180,E1 20217.673,E2 20217.673} C_VEL
LIN {X 0,Y 540.809,Z 681.249,A -85,B 0,C 180,E1 20214.432,E2 20214.432} C_VEL
LIN {X 0,Y 541.453,Z 606.467,A -85,B 0,C 180,E1 20213.279,E2 20213.279} C_VEL
LIN {X 0,Y 538.075,Z 590.422,A -85,B 0,C 180,E1 20212.715,E2 20212.715} C_VEL
LIN {X 0,Y 539.966,Z 550.97,A -85,B 0,C 180,E1 20209.322,E2 20209.322} C_VEL
LIN {X 0,Y 540.088,Z 544.493,A -85,B 0,C 180,E1 20208.731,E2 20208.731} C_VEL
LIN {X 0,Y 533.29,Z 528.447,A -85,B 0,C 180,E1 20206.517,E2 20206.517} C_VEL
LIN {X 0,Y 528.524,Z 517.462,A -85,B 0,C 180,E1 20204.863,E2 20204.863} C_VEL
LIN {X 0,Y 528.461,Z 517.17,A -85,B 0,C 180,E1 20201.964,E2 20201.964} C_VEL
LIN {X 0,Y 528.491,Z 517.211,A -85,B 0,C 180,E1 20198.614,E2 20198.614} C_VEL
LIN {X 0,Y 528.534,Z 517.477,A -85,B 0,C 180,E1 20196.55,E2 20196.55} C_VEL
LIN {X 0,Y 534.869,Z 536.824,A -85,B 0,C 180,E1 20194.572,E2 20194.572} C_VEL
LIN {X 0,Y 534.34,Z 574.647,A -85,B 0,C 180,E1 20191.597,E2 20191.597} C_VEL
LIN {X 0,Y 533.549,Z 615.667,A -85,B 0,C 180,E1 20188.363,E2 20188.363} C_VEL
LIN {X 0,Y 532.586,Z 655.793,A -85,B 0,C 180,E1 20185.191,E2 20185.191} C_VEL
LIN {X 0,Y 531.429,Z 698.993,A -85,B 0,C 180,E1 20181.756,E2 20181.756} C_VEL
LIN {X 0,Y 531.285,Z 705.715,A -85,B 0,C 180,E1 20181.253,E2 20181.253} C_VEL
LIN {X 0,Y 532.506,Z 716.478,A -85,B 0,C 180,E1 20181.049,E2 20181.049} C_VEL
LIN {X 0,Y 531.571,Z 875.803,A -85,B 0,C 180,E1 20178.814,E2 20178.814} C_VEL
LIN {X 0,Y 531.278,Z 892.781,A -85,B 0,C 180,E1 20178.379,E2 20178.379} C_VEL
LIN {X 0,Y 530.896,Z 909.358,A -85,B 0,C 180,E1 20177.765,E2 20177.765} C_VEL
LIN {X 0,Y 530.423,Z 926.181,A -85,B 0,C 180,E1 20176.915,E2 20176.915} C_VEL
LIN {X 0,Y 529.898,Z 942.001,A -85,B 0,C 180,E1 20175.879,E2 20175.879} C_VEL
LIN {X 0,Y 529.41,Z 956.782,A -85,B 0,C 180,E1 20174.66,E2 20174.66} C_VEL
LIN {X 0,Y 528.973,Z 969.853,A -85,B 0,C 180,E1 20173.333,E2 20173.333} C_VEL
LIN {X 0,Y 528.61,Z 981.448,A -85,B 0,C 180,E1 20171.898,E2 20171.898} C_VEL
LIN {X 0,Y 528.309,Z 992.422,A -85,B 0,C 180,E1 20170.219,E2 20170.219} C_VEL
LIN {X 0,Y 528.11,Z 1001.368,A -85,B 0,C 180,E1 20168.493,E2 20168.493} C_VEL
LIN {X 0,Y 527.996,Z 1008.442,A -85,B 0,C 180,E1 20166.743,E2 20166.743} C_VEL
LIN {X 0,Y 527.937,Z 1013.983,A -85,B 0,C 180,E1 20164.889,E2 20164.889} C_VEL
LIN {X 0,Y 527.917,Z 1017.821,A -85,B 0,C 180,E1 20162.932,E2 20162.932} C_VEL
LIN {X 0,Y 527.915,Z 1019.666,A -85,B 0,C 180,E1 20161.086,E2 20161.086} C_VEL
LIN {X 0,Y 527.916,Z 1019.836,A -85,B 0,C 180,E1 20159.349,E2 20159.349} C_VEL
LIN {X 0,Y 527.911,Z 1018.644,A -85,B 0,C 180,E1 20157.612,E2 20157.612} C_VEL
LIN {X 0,Y 527.924,Z 1015.681,A -85,B 0,C 180,E1 20155.764,E2 20155.764} C_VEL
LIN {X 0,Y 527.96,Z 1011.183,A -85,B 0,C 180,E1 20154.022,E2 20154.022} C_VEL
LIN {X 0,Y 528.028,Z 1005.878,A -85,B 0,C 180,E1 20152.493,E2 20152.493} C_VEL
LIN {X 0,Y 528.134,Z 999.662,A -85,B 0,C 180,E1 20151.07,E2 20151.07} C_VEL
LIN {X 0,Y 528.329,Z 991.471,A -85,B 0,C 180,E1 20149.533,E2 20149.533} C_VEL
LIN {X 0,Y 528.633,Z 980.429,A -85,B 0,C 180,E1 20147.881,E2 20147.881} C_VEL
LIN {X 0,Y 528.971,Z 969.577,A -85,B 0,C 180,E1 20146.556,E2 20146.556} C_VEL
LIN {X 0,Y 529.343,Z 958.501,A -85,B 0,C 180,E1 20145.418,E2 20145.418} C_VEL
LIN {X 0,Y 529.819,Z 944.669,A -85,B 0,C 180,E1 20144.232,E2 20144.232} C_VEL
LIN {X 0,Y 530.282,Z 930.025,A -85,B 0,C 180,E1 20143.233,E2 20143.233} C_VEL
LIN {X 0,Y 530.662,Z 916.998,A -85,B 0,C 180,E1 20142.511,E2 20142.511} C_VEL
LIN {X 0,Y 531.061,Z 902.634,A -85,B 0,C 180,E1 20141.873,E2 20141.873} C_VEL
LIN {X 0,Y 531.424,Z 884.849,A -85,B 0,C 180,E1 20141.305,E2 20141.305} C_VEL
LIN {X 0,Y 531.641,Z 868.268,A -85,B 0,C 180,E1 20140.967,E2 20140.967} C_VEL
LIN {X 0,Y 532.342,Z 713.307,A -85,B 0,C 180,E1 20138.809,E2 20138.809} C_VEL
LIN {X 0,Y 531.248,Z 705.087,A -85,B 0,C 180,E1 20138.628,E2 20138.628} C_VEL
LIN {X 0,Y 532.356,Z 666.169,A -85,B 0,C 180,E1 20135.535,E2 20135.535} C_VEL
LIN {X 0,Y 532.994,Z 631.656,A -85,B 0,C 180,E1 20132.881,E2 20132.881} C_VEL
LIN {X 0,Y 533.185,Z 596.838,A -85,B 0,C 180,E1 20130.326,E2 20130.326} C_VEL
LIN {X 0,Y 532.896,Z 565.104,A -85,B 0,C 180,E1 20128.118,E2 20128.118} C_VEL
LIN {X 0,Y 532.259,Z 535.142,A -85,B 0,C 180,E1 20126.177,E2 20126.177} C_VEL
LIN {X 0,Y 531.859,Z 530.975,A -85,B 0,C 180,E1 20125.906,E2 20125.906} C_VEL
LIN {X 0,Y 528.581,Z 517.647,A -85,B 0,C 180,E1 20124.958,E2 20124.958} C_VEL
LIN {X 0,Y 528.496,Z 517.219,A -85,B 0,C 180,E1 20124.759,E2 20124.759} C_VEL
LIN {X 0,Y 528.523,Z 517.194,A -85,B 0,C 180,E1 20121.37,E2 20121.37} C_VEL
LIN {X 0,Y 528.508,Z 517.214,A -85,B 0,C 180,E1 20117.955,E2 20117.955} C_VEL
LIN {X 0,Y 528.567,Z 517.502,A -85,B 0,C 180,E1 20116.634,E2 20116.634} C_VEL
LIN {X 0,Y 530.038,Z 520.987,A -85,B 0,C 180,E1 20116.104,E2 20116.104} C_VEL
LIN {X 0,Y 539.56,Z 541.751,A -85,B 0,C 180,E1 20113.259,E2 20113.259} C_VEL
LIN {X 0,Y 540.968,Z 544.506,A -85,B 0,C 180,E1 20112.953,E2 20112.953} C_VEL
LIN {X 0,Y 542.733,Z 547.825,A -85,B 0,C 180,E1 20112.737,E2 20112.737} C_VEL
LIN {X 0,Y 545.958,Z 563.005,A -85,B 0,C 180,E1 20112.166,E2 20112.166} C_VEL
LIN {X 0,Y 543.317,Z 771.736,A -85,B 0,C 180,E1 20108.856,E2 20108.856} C_VEL
LIN {X 0,Y 541.8,Z 892.419,A -85,B 0,C 180,E1 20106.961,E2 20106.961} C_VEL
LIN {X 0,Y 541.06,Z 915.61,A -85,B 0,C 180,E1 20106.409,E2 20106.409} C_VEL
LIN {X 0,Y 540.186,Z 937.313,A -85,B 0,C 180,E1 20105.711,E2 20105.711} C_VEL
LIN {X 0,Y 539.158,Z 958.388,A -85,B 0,C 180,E1 20104.833,E2 20104.833} C_VEL
LIN {X 0,Y 538.07,Z 978.214,A -85,B 0,C 180,E1 20103.837,E2 20103.837} C_VEL
LIN {X 0,Y 536.753,Z 999.24,A -85,B 0,C 180,E1 20102.571,E2 20102.571} C_VEL
LIN {X 0,Y 535.49,Z 1019.406,A -85,B 0,C 180,E1 20101.145,E2 20101.145} C_VEL
LIN {X 0,Y 534.11,Z 1039.271,A -85,B 0,C 180,E1 20099.495,E2 20099.495} C_VEL
LIN {X 0,Y 532.814,Z 1058.789,A -85,B 0,C 180,E1 20097.614,E2 20097.614} C_VEL
LIN {X 0,Y 531.724,Z 1075.659,A -85,B 0,C 180,E1 20095.746,E2 20095.746} C_VEL
LIN {X 0,Y 530.695,Z 1091.993,A -85,B 0,C 180,E1 20093.66,E2 20093.66} C_VEL
LIN {X 0,Y 529.868,Z 1106.925,A -85,B 0,C 180,E1 20091.474,E2 20091.474} C_VEL
LIN {X 0,Y 529.228,Z 1119.728,A -85,B 0,C 180,E1 20089.307,E2 20089.307} C_VEL
LIN {X 0,Y 528.698,Z 1132.052,A -85,B 0,C 180,E1 20086.878,E2 20086.878} C_VEL
LIN {X 0,Y 528.362,Z 1141.99,A -85,B 0,C 180,E1 20084.577,E2 20084.577} C_VEL
LIN {X 0,Y 528.117,Z 1150.7,A -85,B 0,C 180,E1 20082.131,E2 20082.131} C_VEL
LIN {X 0,Y 527.982,Z 1157.473,A -85,B 0,C 180,E1 20079.813,E2 20079.813} C_VEL
LIN {X 0,Y 527.92,Z 1162.841,A -85,B 0,C 180,E1 20077.4,E2 20077.4} C_VEL
LIN {X 0,Y 527.915,Z 1166.436,A -85,B 0,C 180,E1 20075.216,E2 20075.216} C_VEL
LIN {X 0,Y 527.909,Z 1169.056,A -85,B 0,C 180,E1 20072.605,E2 20072.605} C_VEL
LIN {X 0,Y 527.891,Z 1169.939,A -85,B 0,C 180,E1 20070.326,E2 20070.326} C_VEL
LIN {X 0,Y 527.913,Z 1169.324,A -85,B 0,C 180,E1 20067.829,E2 20067.829} C_VEL
LIN {X 0,Y 527.909,Z 1167.389,A -85,B 0,C 180,E1 20065.546,E2 20065.546} C_VEL
LIN {X 0,Y 527.91,Z 1163.667,A -85,B 0,C 180,E1 20063.038,E2 20063.038} C_VEL
LIN {X 0,Y 527.986,Z 1159.062,A -85,B 0,C 180,E1 20060.847,E2 20060.847} C_VEL
LIN {X 0,Y 528.102,Z 1152.117,A -85,B 0,C 180,E1 20058.312,E2 20058.312} C_VEL
LIN {X 0,Y 528.269,Z 1144.522,A -85,B 0,C 180,E1 20056.091,E2 20056.091} C_VEL
LIN {X 0,Y 528.602,Z 1134.396,A -85,B 0,C 180,E1 20053.63,E2 20053.63} C_VEL
LIN {X 0,Y 529.043,Z 1123.407,A -85,B 0,C 180,E1 20051.373,E2 20051.373} C_VEL
LIN {X 0,Y 529.662,Z 1110.461,A -85,B 0,C 180,E1 20049.097,E2 20049.097} C_VEL
LIN {X 0,Y 530.476,Z 1096.055,A -85,B 0,C 180,E1 20046.895,E2 20046.895} C_VEL
LIN {X 0,Y 531.416,Z 1080.307,A -85,B 0,C 180,E1 20044.822,E2 20044.822} C_VEL
LIN {X 0,Y 532.573,Z 1062.117,A -85,B 0,C 180,E1 20042.736,E2 20042.736} C_VEL
LIN {X 0,Y 533.84,Z 1043.9,A -85,B 0,C 180,E1 20040.92,E2 20040.92} C_VEL
LIN {X 0,Y 535.097,Z 1024.562,A -85,B 0,C 180,E1 20039.264,E2 20039.264} C_VEL
LIN {X 0,Y 536.496,Z 1003.726,A -85,B 0,C 180,E1 20037.727,E2 20037.727} C_VEL
LIN {X 0,Y 537.71,Z 983.812,A -85,B 0,C 180,E1 20036.477,E2 20036.477} C_VEL
LIN {X 0,Y 538.962,Z 962.242,A -85,B 0,C 180,E1 20035.347,E2 20035.347} C_VEL
LIN {X 0,Y 539.936,Z 942.974,A -85,B 0,C 180,E1 20034.511,E2 20034.511} C_VEL
LIN {X 0,Y 540.91,Z 919.206,A -85,B 0,C 180,E1 20033.693,E2 20033.693} C_VEL
LIN {X 0,Y 541.651,Z 897.75,A -85,B 0,C 180,E1 20033.147,E2 20033.147} C_VEL
LIN {X 0,Y 542.21,Z 865.387,A -85,B 0,C 180,E1 20032.595,E2 20032.595} C_VEL
LIN {X 0,Y 544.764,Z 655.366,A -85,B 0,C 180,E1 20029.313,E2 20029.313} C_VEL
LIN {X 0,Y 545.872,Z 558.513,A -85,B 0,C 180,E1 20027.748,E2 20027.748} C_VEL
LIN {X 0,Y 543.617,Z 546.885,A -85,B 0,C 180,E1 20027.328,E2 20027.328} C_VEL
LIN {X 0,Y 540.567,Z 542.004,A -85,B 0,C 180,E1 20026.937,E2 20026.937} C_VEL
LIN {X 0,Y 530.321,Z 521.344,A -85,B 0,C 180,E1 20024.385,E2 20024.385} C_VEL
LIN {X 0,Y 528.589,Z 517.692,A -85,B 0,C 180,E1 20023.896,E2 20023.896} C_VEL
LIN {X 0,Y 528.52,Z 517.192,A -85,B 0,C 180,E1 20023.52,E2 20023.52} C_VEL
LIN {X 0,Y 528.517,Z 517.199,A -85,B 0,C 180,E1 20019.987,E2 20019.987} C_VEL
LIN {X 0,Y 528.505,Z 517.193,A -85,B 0,C 180,E1 20016.579,E2 20016.579} C_VEL
LIN {X 0,Y 528.51,Z 517.199,A -85,B 0,C 180,E1 20013.259,E2 20013.259} C_VEL
LIN {X 0,Y 528.515,Z 517.215,A -85,B 0,C 180,E1 20009.838,E2 20009.838} C_VEL
LIN {X 0,Y 528.516,Z 517.198,A -85,B 0,C 180,E1 20006.269,E2 20006.269} C_VEL
LIN {X 0,Y 528.509,Z 517.198,A -85,B 0,C 180,E1 20002.819,E2 20002.819} C_VEL
LIN {X 0,Y 528.51,Z 517.208,A -85,B 0,C 180,E1 19999.448,E2 19999.448} C_VEL
LIN {X 0,Y 528.518,Z 517.19,A -85,B 0,C 180,E1 19996.033,E2 19996.033} C_VEL
LIN {X 0,Y 528.517,Z 517.215,A -85,B 0,C 180,E1 19992.53,E2 19992.53} C_VEL
LIN {X 0,Y 528.51,Z 517.191,A -85,B 0,C 180,E1 19989.144,E2 19989.144} C_VEL
LIN {X 0,Y 528.509,Z 517.211,A -85,B 0,C 180,E1 19985.754,E2 19985.754} C_VEL
LIN {X 0,Y 528.52,Z 517.211,A -85,B 0,C 180,E1 19982.277,E2 19982.277} C_VEL
LIN {X 0,Y 528.521,Z 517.206,A -85,B 0,C 180,E1 19978.807,E2 19978.807} C_VEL
LIN {X 0,Y 528.505,Z 517.213,A -85,B 0,C 180,E1 19975.334,E2 19975.334} C_VEL
LIN {X 0,Y 528.514,Z 517.207,A -85,B 0,C 180,E1 19971.952,E2 19971.952} C_VEL
LIN {X 0,Y 528.515,Z 517.195,A -85,B 0,C 180,E1 19968.513,E2 19968.513} C_VEL
LIN {X 0,Y 528.51,Z 517.215,A -85,B 0,C 180,E1 19964.978,E2 19964.978} C_VEL
LIN {X 0,Y 528.514,Z 517.197,A -85,B 0,C 180,E1 19961.582,E2 19961.582} C_VEL
LIN {X 0,Y 528.504,Z 517.212,A -85,B 0,C 180,E1 19958.234,E2 19958.234} C_VEL
LIN {X 0,Y 528.518,Z 517.192,A -85,B 0,C 180,E1 19954.807,E2 19954.807} C_VEL
LIN {X 0,Y 528.526,Z 517.21,A -85,B 0,C 180,E1 19951.281,E2 19951.281} C_VEL
LIN {X 0,Y 528.501,Z 517.206,A -85,B 0,C 180,E1 19947.885,E2 19947.885} C_VEL
LIN {X 0,Y 528.516,Z 517.195,A -85,B 0,C 180,E1 19944.438,E2 19944.438} C_VEL
LIN {X 0,Y 528.503,Z 517.214,A -85,B 0,C 180,E1 19941.662,E2 19941.662} C_VEL
LIN {X 0,Y 527.496,Z 517.333,A -85,B 0,C 180,E1 19940.827,E2 19940.827} C_VEL
LIN {X 0,Y 521.106,Z 518.134,A -85,B 0,C 180,E1 19938.48,E2 19938.48} C_VEL
LIN {X 0,Y 520.583,Z 518.205,A -85,B 0,C 180,E1 19937.869,E2 19937.869} C_VEL
LIN {X 0,Y 520.612,Z 518.437,A -85,B 0,C 180,E1 19934.598,E2 19934.598} C_VEL
LIN {X 0,Y 522.023,Z 521.886,A -85,B 0,C 180,E1 19934.089,E2 19934.089} C_VEL
LIN {X 0,Y 530.149,Z 538.644,A -85,B 0,C 180,E1 19931.843,E2 19931.843} C_VEL
LIN {X 0,Y 534.464,Z 548.694,A -85,B 0,C 180,E1 19930.619,E2 19930.619} C_VEL
LIN {X 0,Y 532.449,Z 589.458,A -85,B 0,C 180,E1 19927.681,E2 19927.681} C_VEL
LIN {X 0,Y 535.233,Z 607.413,A -85,B 0,C 180,E1 19927.113,E2 19927.113} C_VEL
LIN {X 0,Y 532.481,Z 839.769,A -85,B 0,C 180,E1 19923.567,E2 19923.567} C_VEL
LIN {X 0,Y 531.758,Z 897.35,A -85,B 0,C 180,E1 19922.667,E2 19922.667} C_VEL
LIN {X 0,Y 531.034,Z 919.018,A -85,B 0,C 180,E1 19922.13,E2 19922.13} C_VEL
LIN {X 0,Y 530.2,Z 940.402,A -85,B 0,C 180,E1 19921.397,E2 19921.397} C_VEL
LIN {X 0,Y 529.219,Z 960.678,A -85,B 0,C 180,E1 19920.511,E2 19920.511} C_VEL
LIN {X 0,Y 528.09,Z 980.469,A -85,B 0,C 180,E1 19919.432,E2 19919.432} C_VEL
LIN {X 0,Y 526.834,Z 1001.039,A -85,B 0,C 180,E1 19918.078,E2 19918.078} C_VEL
LIN {X 0,Y 525.661,Z 1019.671,A -85,B 0,C 180,E1 19916.621,E2 19916.621} C_VEL
LIN {X 0,Y 524.483,Z 1037.56,A -85,B 0,C 180,E1 19914.978,E2 19914.978} C_VEL
LIN {X 0,Y 523.433,Z 1053.664,A -85,B 0,C 180,E1 19913.248,E2 19913.248} C_VEL
LIN {X 0,Y 522.45,Z 1069.734,A -85,B 0,C 180,E1 19911.249,E2 19911.249} C_VEL
LIN {X 0,Y 521.682,Z 1083.566,A -85,B 0,C 180,E1 19909.248,E2 19909.248} C_VEL
LIN {X 0,Y 521.053,Z 1096.016,A -85,B 0,C 180,E1 19907.133,E2 19907.133} C_VEL
LIN {X 0,Y 520.586,Z 1107.114,A -85,B 0,C 180,E1 19904.914,E2 19904.914} C_VEL
LIN {X 0,Y 520.277,Z 1116.593,A -85,B 0,C 180,E1 19902.655,E2 19902.655} C_VEL
LIN {X 0,Y 520.088,Z 1124.24,A -85,B 0,C 180,E1 19900.411,E2 19900.411} C_VEL
LIN {X 0,Y 519.975,Z 1130.726,A -85,B 0,C 180,E1 19897.989,E2 19897.989} C_VEL
LIN {X 0,Y 519.926,Z 1135.418,A -85,B 0,C 180,E1 19895.628,E2 19895.628} C_VEL
LIN {X 0,Y 519.91,Z 1138.353,A -85,B 0,C 180,E1 19893.307,E2 19893.307} C_VEL
LIN {X 0,Y 519.904,Z 1139.817,A -85,B 0,C 180,E1 19890.882,E2 19890.882} C_VEL
LIN {X 0,Y 519.903,Z 1139.723,A -85,B 0,C 180,E1 19888.567,E2 19888.567} C_VEL
LIN {X 0,Y 519.906,Z 1137.995,A -85,B 0,C 180,E1 19886.251,E2 19886.251} C_VEL
LIN {X 0,Y 519.932,Z 1134.6,A -85,B 0,C 180,E1 19883.818,E2 19883.818} C_VEL
LIN {X 0,Y 519.993,Z 1129.731,A -85,B 0,C 180,E1 19881.486,E2 19881.486} C_VEL
LIN {X 0,Y 520.11,Z 1123.11,A -85,B 0,C 180,E1 19879.141,E2 19879.141} C_VEL
LIN {X 0,Y 520.338,Z 1114.741,A -85,B 0,C 180,E1 19876.781,E2 19876.781} C_VEL
LIN {X 0,Y 520.687,Z 1104.927,A -85,B 0,C 180,E1 19874.519,E2 19874.519} C_VEL
LIN {X 0,Y 521.159,Z 1093.665,A -85,B 0,C 180,E1 19872.354,E2 19872.354} C_VEL
LIN {X 0,Y 521.845,Z 1080.353,A -85,B 0,C 180,E1 19870.176,E2 19870.176} C_VEL
LIN {X 0,Y 522.664,Z 1066.431,A -85,B 0,C 180,E1 19868.215,E2 19868.215} C_VEL
LIN {X 0,Y 523.647,Z 1050.467,A -85,B 0,C 180,E1 19866.296,E2 19866.296} C_VEL
LIN {X 0,Y 524.7,Z 1034,A -85,B 0,C 180,E1 19864.588,E2 19864.588} C_VEL
LIN {X 0,Y 525.896,Z 1015.898,A -85,B 0,C 180,E1 19862.974,E2 19862.974} C_VEL
LIN {X 0,Y 527.097,Z 997.35,A -85,B 0,C 180,E1 19861.567,E2 19861.567} C_VEL
LIN {X 0,Y 528.231,Z 977.801,A -85,B 0,C 180,E1 19860.321,E2 19860.321} C_VEL
LIN {X 0,Y 529.412,Z 956.737,A -85,B 0,C 180,E1 19859.215,E2 19859.215} C_VEL
LIN {X 0,Y 530.382,Z 936.578,A -85,B 0,C 180,E1 19858.362,E2 19858.362} C_VEL
LIN {X 0,Y 531.168,Z 915.578,A -85,B 0,C 180,E1 19857.683,E2 19857.683} C_VEL
LIN {X 0,Y 531.819,Z 893.489,A -85,B 0,C 180,E1 19857.173,E2 19857.173} C_VEL
LIN {X 0,Y 534.331,Z 679.026,A -85,B 0,C 180,E1 19853.898,E2 19853.898} C_VEL
LIN {X 0,Y 535,Z 608.057,A -85,B 0,C 180,E1 19852.788,E2 19852.788} C_VEL
LIN {X 0,Y 531.381,Z 590.262,A -85,B 0,C 180,E1 19852.129,E2 19852.129} C_VEL
LIN {X 0,Y 533.424,Z 551.819,A -85,B 0,C 180,E1 19848.78,E2 19848.78} C_VEL
LIN {X 0,Y 533.389,Z 548.119,A -85,B 0,C 180,E1 19848.426,E2 19848.426} C_VEL
LIN {X 0,Y 526.954,Z 532.981,A -85,B 0,C 180,E1 19846.296,E2 19846.296} C_VEL
LIN {X 0,Y 522.1,Z 522.074,A -85,B 0,C 180,E1 19844.655,E2 19844.655} C_VEL
LIN {X 0,Y 520.558,Z 518.404,A -85,B 0,C 180,E1 19844.043,E2 19844.043} C_VEL
LIN {X 0,Y 520.584,Z 518.164,A -85,B 0,C 180,E1 19841.061,E2 19841.061} C_VEL
LIN {X 0,Y 520.523,Z 518.201,A -85,B 0,C 180,E1 19837.79,E2 19837.79} C_VEL
LIN {X 0,Y 520.637,Z 518.549,A -85,B 0,C 180,E1 19836.966,E2 19836.966} C_VEL
LIN {X 0,Y 527.615,Z 539.558,A -85,B 0,C 180,E1 19834.809,E2 19834.809} C_VEL
LIN {X 0,Y 526.96,Z 580.247,A -85,B 0,C 180,E1 19831.576,E2 19831.576} C_VEL
LIN {X 0,Y 526.054,Z 620.642,A -85,B 0,C 180,E1 19828.371,E2 19828.371} C_VEL
LIN {X 0,Y 525.009,Z 661.375,A -85,B 0,C 180,E1 19825.132,E2 19825.132} C_VEL
LIN {X 0,Y 523.769,Z 704.606,A -85,B 0,C 180,E1 19821.678,E2 19821.678} C_VEL
LIN {X 0,Y 523.828,Z 707.044,A -85,B 0,C 180,E1 19821.533,E2 19821.533} C_VEL
LIN {X 0,Y 524.982,Z 717.412,A -85,B 0,C 180,E1 19821.334,E2 19821.334} C_VEL
LIN {X 0,Y 524,Z 875.606,A -85,B 0,C 180,E1 19819.1,E2 19819.1} C_VEL
LIN {X 0,Y 523.681,Z 892.566,A -85,B 0,C 180,E1 19818.662,E2 19818.662} C_VEL
LIN {X 0,Y 523.276,Z 908.689,A -85,B 0,C 180,E1 19818.064,E2 19818.064} C_VEL
LIN {X 0,Y 522.738,Z 925.902,A -85,B 0,C 180,E1 19817.189,E2 19817.189} C_VEL
LIN {X 0,Y 522.147,Z 942.008,A -85,B 0,C 180,E1 19816.121,E2 19816.121} C_VEL
LIN {X 0,Y 521.601,Z 956.789,A -85,B 0,C 180,E1 19814.884,E2 19814.884} C_VEL
LIN {X 0,Y 521.11,Z 969.857,A -85,B 0,C 180,E1 19813.538,E2 19813.538} C_VEL
LIN {X 0,Y 520.702,Z 981.453,A -85,B 0,C 180,E1 19812.082,E2 19812.082} C_VEL
LIN {X 0,Y 520.367,Z 992.258,A -85,B 0,C 180,E1 19810.406,E2 19810.406} C_VEL
LIN {X 0,Y 520.137,Z 1001.371,A -85,B 0,C 180,E1 19808.624,E2 19808.624} C_VEL
LIN {X 0,Y 520.007,Z 1008.442,A -85,B 0,C 180,E1 19806.847,E2 19806.847} C_VEL
LIN {X 0,Y 519.941,Z 1013.985,A -85,B 0,C 180,E1 19804.965,E2 19804.965} C_VEL
LIN {X 0,Y 519.917,Z 1017.823,A -85,B 0,C 180,E1 19802.977,E2 19802.977} C_VEL
LIN {X 0,Y 519.916,Z 1019.665,A -85,B 0,C 180,E1 19801.102,E2 19801.102} C_VEL
LIN {X 0,Y 519.916,Z 1019.829,A -85,B 0,C 180,E1 19799.339,E2 19799.339} C_VEL
LIN {X 0,Y 519.912,Z 1018.641,A -85,B 0,C 180,E1 19797.575,E2 19797.575} C_VEL
LIN {X 0,Y 519.926,Z 1015.68,A -85,B 0,C 180,E1 19795.699,E2 19795.699} C_VEL
LIN {X 0,Y 519.966,Z 1011.175,A -85,B 0,C 180,E1 19793.929,E2 19793.929} C_VEL
LIN {X 0,Y 520.045,Z 1005.867,A -85,B 0,C 180,E1 19792.377,E2 19792.377} C_VEL
LIN {X 0,Y 520.165,Z 999.652,A -85,B 0,C 180,E1 19790.932,E2 19790.932} C_VEL
LIN {X 0,Y 520.387,Z 991.465,A -85,B 0,C 180,E1 19789.371,E2 19789.371} C_VEL
LIN {X 0,Y 520.73,Z 980.416,A -85,B 0,C 180,E1 19787.694,E2 19787.694} C_VEL
LIN {X 0,Y 521.091,Z 970.058,A -85,B 0,C 180,E1 19786.406,E2 19786.406} C_VEL
LIN {X 0,Y 521.489,Z 959.391,A -85,B 0,C 180,E1 19785.283,E2 19785.283} C_VEL
LIN {X 0,Y 521.948,Z 947.376,A -85,B 0,C 180,E1 19784.216,E2 19784.216} C_VEL
LIN {X 0,Y 522.518,Z 931.863,A -85,B 0,C 180,E1 19783.091,E2 19783.091} C_VEL
LIN {X 0,Y 522.963,Z 918.096,A -85,B 0,C 180,E1 19782.303,E2 19782.303} C_VEL
LIN {X 0,Y 523.392,Z 903.976,A -85,B 0,C 180,E1 19781.656,E2 19781.656} C_VEL
LIN {X 0,Y 523.803,Z 886.836,A -85,B 0,C 180,E1 19781.076,E2 19781.076} C_VEL
LIN {X 0,Y 524.034,Z 870.98,A -85,B 0,C 180,E1 19780.73,E2 19780.73} C_VEL
LIN {X 0,Y 524.765,Z 714.202,A -85,B 0,C 180,E1 19778.54,E2 19778.54} C_VEL
LIN {X 0,Y 523.818,Z 706.88,A -85,B 0,C 180,E1 19778.37,E2 19778.37} C_VEL
LIN {X 0,Y 524.899,Z 667.613,A -85,B 0,C 180,E1 19775.262,E2 19775.262} C_VEL
LIN {X 0,Y 525.529,Z 629.239,A -85,B 0,C 180,E1 19772.34,E2 19772.34} C_VEL
LIN {X 0,Y 525.609,Z 594.053,A -85,B 0,C 180,E1 19769.785,E2 19769.785} C_VEL
LIN {X 0,Y 525.212,Z 561.026,A -85,B 0,C 180,E1 19767.531,E2 19767.531} C_VEL
LIN {X 0,Y 524.36,Z 533.494,A -85,B 0,C 180,E1 19765.771,E2 19765.771} C_VEL
LIN {X 0,Y 520.619,Z 518.635,A -85,B 0,C 180,E1 19764.709,E2 19764.709} C_VEL
LIN {X 0,Y 520.538,Z 518.211,A -85,B 0,C 180,E1 19764.409,E2 19764.409} C_VEL
LIN {X 0,Y 520.584,Z 518.172,A -85,B 0,C 180,E1 19761.066,E2 19761.066} C_VEL
LIN {X 0,Y 520.588,Z 518.263,A -85,B 0,C 180,E1 19757.613,E2 19757.613} C_VEL
LIN {X 0,Y 520.682,Z 518.821,A -85,B 0,C 180,E1 19757.381,E2 19757.381} C_VEL
LIN {X 0,Y 528.174,Z 535.036,A -85,B 0,C 180,E1 19755.005,E2 19755.005} C_VEL
LIN {X 0,Y 532.631,Z 544.715,A -85,B 0,C 180,E1 19753.721,E2 19753.721} C_VEL
LIN {X 0,Y 537.123,Z 552.012,A -85,B 0,C 180,E1 19753.168,E2 19753.168} C_VEL
LIN {X 0,Y 539.911,Z 564.905,A -85,B 0,C 180,E1 19752.696,E2 19752.696} C_VEL
LIN {X 0,Y 537.155,Z 766.901,A -85,B 0,C 180,E1 19749.47,E2 19749.47} C_VEL
LIN {X 0,Y 535.404,Z 892.337,A -85,B 0,C 180,E1 19747.479,E2 19747.479} C_VEL
LIN {X 0,Y 534.609,Z 915.348,A -85,B 0,C 180,E1 19746.929,E2 19746.929} C_VEL
LIN {X 0,Y 533.669,Z 936.454,A -85,B 0,C 180,E1 19746.248,E2 19746.248} C_VEL
LIN {X 0,Y 532.488,Z 958.384,A -85,B 0,C 180,E1 19745.334,E2 19745.334} C_VEL
LIN {X 0,Y 531.275,Z 978.571,A -85,B 0,C 180,E1 19744.309,E2 19744.309} C_VEL
LIN {X 0,Y 529.771,Z 1000.137,A -85,B 0,C 180,E1 19742.991,E2 19742.991} C_VEL
LIN {X 0,Y 528.373,Z 1020.184,A -85,B 0,C 180,E1 19741.549,E2 19741.549} C_VEL
LIN {X 0,Y 526.894,Z 1039.269,A -85,B 0,C 180,E1 19739.939,E2 19739.939} C_VEL
LIN {X 0,Y 525.422,Z 1059.137,A -85,B 0,C 180,E1 19737.998,E2 19737.998} C_VEL
LIN {X 0,Y 524.213,Z 1075.659,A -85,B 0,C 180,E1 19736.142,E2 19736.142} C_VEL
LIN {X 0,Y 523.069,Z 1091.991,A -85,B 0,C 180,E1 19734.026,E2 19734.026} C_VEL
LIN {X 0,Y 522.119,Z 1107.242,A -85,B 0,C 180,E1 19731.756,E2 19731.756} C_VEL
LIN {X 0,Y 521.408,Z 1119.726,A -85,B 0,C 180,E1 19729.608,E2 19729.608} C_VEL
LIN {X 0,Y 520.821,Z 1131.804,A -85,B 0,C 180,E1 19727.196,E2 19727.196} C_VEL
LIN {X 0,Y 520.44,Z 1141.577,A -85,B 0,C 180,E1 19724.907,E2 19724.907} C_VEL
LIN {X 0,Y 520.155,Z 1150.345,A -85,B 0,C 180,E1 19722.433,E2 19722.433} C_VEL
LIN {X 0,Y 520.018,Z 1156.867,A -85,B 0,C 180,E1 19720.189,E2 19720.189} C_VEL
LIN {X 0,Y 519.94,Z 1162.634,A -85,B 0,C 180,E1 19717.625,E2 19717.625} C_VEL
LIN {X 0,Y 519.908,Z 1166.277,A -85,B 0,C 180,E1 19715.407,E2 19715.407} C_VEL
LIN {X 0,Y 519.893,Z 1168.919,A -85,B 0,C 180,E1 19712.866,E2 19712.866} C_VEL
LIN {X 0,Y 519.884,Z 1169.872,A -85,B 0,C 180,E1 19710.661,E2 19710.661} C_VEL
LIN {X 0,Y 519.906,Z 1169.526,A -85,B 0,C 180,E1 19708.126,E2 19708.126} C_VEL
LIN {X 0,Y 519.914,Z 1167.616,A -85,B 0,C 180,E1 19705.699,E2 19705.699} C_VEL
LIN {X 0,Y 519.917,Z 1164.081,A -85,B 0,C 180,E1 19703.152,E2 19703.152} C_VEL
LIN {X 0,Y 519.991,Z 1159.573,A -85,B 0,C 180,E1 19700.928,E2 19700.928} C_VEL
LIN {X 0,Y 520.104,Z 1153.176,A -85,B 0,C 180,E1 19698.467,E2 19698.467} C_VEL
LIN {X 0,Y 520.297,Z 1145.342,A -85,B 0,C 180,E1 19696.101,E2 19696.101} C_VEL
LIN {X 0,Y 520.645,Z 1135.939,A -85,B 0,C 180,E1 19693.717,E2 19693.717} C_VEL
LIN {X 0,Y 521.119,Z 1125.056,A -85,B 0,C 180,E1 19691.409,E2 19691.409} C_VEL
LIN {X 0,Y 521.829,Z 1111.86,A -85,B 0,C 180,E1 19689.004,E2 19689.004} C_VEL
LIN {X 0,Y 522.648,Z 1098.563,A -85,B 0,C 180,E1 19686.91,E2 19686.91} C_VEL
LIN {X 0,Y 523.704,Z 1082.727,A -85,B 0,C 180,E1 19684.741,E2 19684.741} C_VEL
LIN {X 0,Y 524.928,Z 1065.981,A -85,B 0,C 180,E1 19682.735,E2 19682.735} C_VEL
LIN {X 0,Y 526.239,Z 1048.178,A -85,B 0,C 180,E1 19680.895,E2 19680.895} C_VEL
LIN {X 0,Y 527.725,Z 1028.258,A -85,B 0,C 180,E1 19679.106,E2 19679.106} C_VEL
LIN {X 0,Y 529.164,Z 1009.142,A -85,B 0,C 180,E1 19677.629,E2 19677.629} C_VEL
LIN {X 0,Y 530.627,Z 987.828,A -85,B 0,C 180,E1 19676.229,E2 19676.229} C_VEL
LIN {X 0,Y 532.064,Z 966.064,A -85,B 0,C 180,E1 19675.029,E2 19675.029} C_VEL
LIN {X 0,Y 533.225,Z 945.305,A -85,B 0,C 180,E1 19674.1,E2 19674.1} C_VEL
LIN {X 0,Y 534.286,Z 923.679,A -85,B 0,C 180,E1 19673.313,E2 19673.313} C_VEL
LIN {X 0,Y 535.093,Z 901.321,A -85,B 0,C 180,E1 19672.712,E2 19672.712} C_VEL
LIN {X 0,Y 535.734,Z 875.311,A -85,B 0,C 180,E1 19672.229,E2 19672.229} C_VEL
LIN {X 0,Y 538.594,Z 662.951,A -85,B 0,C 180,E1 19668.878,E2 19668.878} C_VEL
LIN {X 0,Y 539.824,Z 560.236,A -85,B 0,C 180,E1 19667.216,E2 19667.216} C_VEL
LIN {X 0,Y 537.913,Z 551.1,A -85,B 0,C 180,E1 19666.889,E2 19666.889} C_VEL
LIN {X 0,Y 532.517,Z 542.759,A -85,B 0,C 180,E1 19666.214,E2 19666.214} C_VEL
LIN {X 0,Y 523.83,Z 525.491,A -85,B 0,C 180,E1 19664.009,E2 19664.009} C_VEL
LIN {X 0,Y 522.226,Z 522.139,A -85,B 0,C 180,E1 19663.571,E2 19663.571} C_VEL
LIN {X 0,Y 520.614,Z 518.494,A -85,B 0,C 180,E1 19663.052,E2 19663.052} C_VEL
LIN {X 0,Y 520.572,Z 518.181,A -85,B 0,C 180,E1 19660.48,E2 19660.48} C_VEL
LIN {X 0,Y 520.579,Z 518.178,A -85,B 0,C 180,E1 19656.953,E2 19656.953} C_VEL
LIN {X 0,Y 520.574,Z 518.189,A -85,B 0,C 180,E1 19653.451,E2 19653.451} C_VEL
LIN {X 0,Y 520.572,Z 518.203,A -85,B 0,C 180,E1 19649.976,E2 19649.976} C_VEL
LIN {X 0,Y 520.582,Z 518.186,A -85,B 0,C 180,E1 19646.461,E2 19646.461} C_VEL
LIN {X 0,Y 520.572,Z 518.188,A -85,B 0,C 180,E1 19642.948,E2 19642.948} C_VEL
LIN {X 0,Y 520.572,Z 518.195,A -85,B 0,C 180,E1 19639.524,E2 19639.524} C_VEL
LIN {X 0,Y 520.578,Z 518.178,A -85,B 0,C 180,E1 19636.056,E2 19636.056} C_VEL
LIN {X 0,Y 520.578,Z 518.204,A -85,B 0,C 180,E1 19632.535,E2 19632.535} C_VEL
LIN {X 0,Y 520.57,Z 518.177,A -85,B 0,C 180,E1 19629.061,E2 19629.061} C_VEL
LIN {X 0,Y 520.573,Z 518.199,A -85,B 0,C 180,E1 19625.621,E2 19625.621} C_VEL
LIN {X 0,Y 520.581,Z 518.203,A -85,B 0,C 180,E1 19622.091,E2 19622.091} C_VEL
LIN {X 0,Y 520.578,Z 518.196,A -85,B 0,C 180,E1 19618.679,E2 19618.679} C_VEL
LIN {X 0,Y 520.567,Z 518.201,A -85,B 0,C 180,E1 19615.262,E2 19615.262} C_VEL
LIN {X 0,Y 520.579,Z 518.197,A -85,B 0,C 180,E1 19611.829,E2 19611.829} C_VEL
LIN {X 0,Y 520.581,Z 518.183,A -85,B 0,C 180,E1 19608.365,E2 19608.365} C_VEL
LIN {X 0,Y 520.567,Z 518.204,A -85,B 0,C 180,E1 19604.857,E2 19604.857} C_VEL
LIN {X 0,Y 520.577,Z 518.18,A -85,B 0,C 180,E1 19601.407,E2 19601.407} C_VEL
LIN {X 0,Y 520.583,Z 518.198,A -85,B 0,C 180,E1 19597.886,E2 19597.886} C_VEL
LIN {X 0,Y 520.567,Z 518.18,A -85,B 0,C 180,E1 19594.395,E2 19594.395} C_VEL
LIN {X 0,Y 520.579,Z 518.201,A -85,B 0,C 180,E1 19590.916,E2 19590.916} C_VEL
LIN {X 0,Y 520.571,Z 518.198,A -85,B 0,C 180,E1 19587.466,E2 19587.466} C_VEL
LIN {X 0,Y 520.57,Z 518.182,A -85,B 0,C 180,E1 19583.961,E2 19583.961} C_VEL
LIN {X 0,Y 520.579,Z 518.186,A -85,B 0,C 180,E1 19580.525,E2 19580.525} C_VEL
LIN {X 0,Y 520.583,Z 518.205,A -85,B 0,C 180,E1 19577.869,E2 19577.869} C_VEL
LIN {X 0,Y 519.741,Z 518.437,A -85,B 0,C 180,E1 19577.352,E2 19577.352} C_VEL
LIN {X 0,Y 515.557,Z 518.805,A -85,B 0,C 180,E1 19576.394,E2 19576.394} C_VEL
LIN {X 0,Y 512.863,Z 519.17,A -85,B 0,C 180,E1 19575.634,E2 19575.634} C_VEL
LIN {X 0,Y 512.717,Z 519.742,A -85,B 0,C 180,E1 19575.36,E2 19575.36} C_VEL
LIN {X 0,Y 514.455,Z 523.392,A -85,B 0,C 180,E1 19574.815,E2 19574.815} C_VEL
LIN {X 0,Y 523.016,Z 541.232,A -85,B 0,C 180,E1 19572.364,E2 19572.364} C_VEL
LIN {X 0,Y 527.916,Z 552.629,A -85,B 0,C 180,E1 19570.944,E2 19570.944} C_VEL
LIN {X 0,Y 526.015,Z 589.66,A -85,B 0,C 180,E1 19568.265,E2 19568.265} C_VEL
LIN {X 0,Y 529.063,Z 608.931,A -85,B 0,C 180,E1 19567.645,E2 19567.645} C_VEL
LIN {X 0,Y 526.257,Z 805.989,A -85,B 0,C 180,E1 19564.565,E2 19564.565} C_VEL
LIN {X 0,Y 525.044,Z 896.639,A -85,B 0,C 180,E1 19563.155,E2 19563.155} C_VEL
LIN {X 0,Y 524.28,Z 918.13,A -85,B 0,C 180,E1 19562.624,E2 19562.624} C_VEL
LIN {X 0,Y 523.322,Z 940.418,A -85,B 0,C 180,E1 19561.857,E2 19561.857} C_VEL
LIN {X 0,Y 522.29,Z 960.022,A -85,B 0,C 180,E1 19560.995,E2 19560.995} C_VEL
LIN {X 0,Y 521.005,Z 980.432,A -85,B 0,C 180,E1 19559.875,E2 19559.875} C_VEL
LIN {X 0,Y 519.694,Z 1000.235,A -85,B 0,C 180,E1 19558.561,E2 19558.561} C_VEL
LIN {X 0,Y 518.428,Z 1018.442,A -85,B 0,C 180,E1 19557.137,E2 19557.137} C_VEL
LIN {X 0,Y 517.144,Z 1035.758,A -85,B 0,C 180,E1 19555.541,E2 19555.541} C_VEL
LIN {X 0,Y 515.911,Z 1053.018,A -85,B 0,C 180,E1 19553.685,E2 19553.685} C_VEL
LIN {X 0,Y 514.868,Z 1068.355,A -85,B 0,C 180,E1 19551.772,E2 19551.772} C_VEL
LIN {X 0,Y 513.953,Z 1082.844,A -85,B 0,C 180,E1 19549.667,E2 19549.667} C_VEL
LIN {X 0,Y 513.246,Z 1095.077,A -85,B 0,C 180,E1 19547.575,E2 19547.575} C_VEL
LIN {X 0,Y 512.7,Z 1106.599,A -85,B 0,C 180,E1 19545.265,E2 19545.265} C_VEL
LIN {X 0,Y 512.345,Z 1116.189,A -85,B 0,C 180,E1 19542.969,E2 19542.969} C_VEL
LIN {X 0,Y 512.119,Z 1123.888,A -85,B 0,C 180,E1 19540.689,E2 19540.689} C_VEL
LIN {X 0,Y 511.985,Z 1130.545,A -85,B 0,C 180,E1 19538.196,E2 19538.196} C_VEL
LIN {X 0,Y 511.929,Z 1135.253,A -85,B 0,C 180,E1 19535.829,E2 19535.829} C_VEL
LIN {X 0,Y 511.91,Z 1138.241,A -85,B 0,C 180,E1 19533.471,E2 19533.471} C_VEL
LIN {X 0,Y 511.908,Z 1139.794,A -85,B 0,C 180,E1 19531.007,E2 19531.007} C_VEL
LIN {X 0,Y 511.906,Z 1139.745,A -85,B 0,C 180,E1 19528.657,E2 19528.657} C_VEL
LIN {X 0,Y 511.907,Z 1138.107,A -85,B 0,C 180,E1 19526.304,E2 19526.304} C_VEL
LIN {X 0,Y 511.932,Z 1135.011,A -85,B 0,C 180,E1 19523.946,E2 19523.946} C_VEL
LIN {X 0,Y 511.993,Z 1130.238,A -85,B 0,C 180,E1 19521.578,E2 19521.578} C_VEL
LIN {X 0,Y 512.126,Z 1123.594,A -85,B 0,C 180,E1 19519.126,E2 19519.126} C_VEL
LIN {X 0,Y 512.366,Z 1115.657,A -85,B 0,C 180,E1 19516.802,E2 19516.802} C_VEL
LIN {X 0,Y 512.736,Z 1105.963,A -85,B 0,C 180,E1 19514.505,E2 19514.505} C_VEL
LIN {X 0,Y 513.29,Z 1094.295,A -85,B 0,C 180,E1 19512.192,E2 19512.192} C_VEL
LIN {X 0,Y 514.046,Z 1081.118,A -85,B 0,C 180,E1 19509.981,E2 19509.981} C_VEL
LIN {X 0,Y 514.939,Z 1067.289,A -85,B 0,C 180,E1 19507.991,E2 19507.991} C_VEL
LIN {X 0,Y 515.982,Z 1052.024,A -85,B 0,C 180,E1 19506.109,E2 19506.109} C_VEL
LIN {X 0,Y 517.259,Z 1034.219,A -85,B 0,C 180,E1 19504.219,E2 19504.219} C_VEL
LIN {X 0,Y 518.539,Z 1016.619,A -85,B 0,C 180,E1 19502.62,E2 19502.62} C_VEL
LIN {X 0,Y 519.855,Z 998.149,A -85,B 0,C 180,E1 19501.197,E2 19501.197} C_VEL
LIN {X 0,Y 521.12,Z 978.495,A -85,B 0,C 180,E1 19499.92,E2 19499.92} C_VEL
LIN {X 0,Y 522.395,Z 958.041,A -85,B 0,C 180,E1 19498.821,E2 19498.821} C_VEL
LIN {X 0,Y 523.437,Z 938.112,A -85,B 0,C 180,E1 19497.96,E2 19497.96} C_VEL
LIN {X 0,Y 524.336,Z 916.789,A -85,B 0,C 180,E1 19497.248,E2 19497.248} C_VEL
LIN {X 0,Y 525.063,Z 895.422,A -85,B 0,C 180,E1 19496.733,E2 19496.733} C_VEL
LIN {X 0,Y 528.196,Z 662.981,A -85,B 0,C 180,E1 19493.125,E2 19493.125} C_VEL
LIN {X 0,Y 528.826,Z 609.766,A -85,B 0,C 180,E1 19492.26,E2 19492.26} C_VEL
LIN {X 0,Y 524.736,Z 589.603,A -85,B 0,C 180,E1 19491.493,E2 19491.493} C_VEL
LIN {X 0,Y 526.946,Z 552.404,A -85,B 0,C 180,E1 19488.199,E2 19488.199} C_VEL
LIN {X 0,Y 520.279,Z 536.716,A -85,B 0,C 180,E1 19485.951,E2 19485.951} C_VEL
LIN {X 0,Y 515.406,Z 526.048,A -85,B 0,C 180,E1 19484.297,E2 19484.297} C_VEL
LIN {X 0,Y 512.677,Z 519.394,A -85,B 0,C 180,E1 19483.209,E2 19483.209} C_VEL
LIN {X 0,Y 512.582,Z 519.19,A -85,B 0,C 180,E1 19480.069,E2 19480.069} C_VEL
LIN {X 0,Y 512.644,Z 519.469,A -85,B 0,C 180,E1 19477.43,E2 19477.43} C_VEL
LIN {X 0,Y 520.315,Z 542.209,A -85,B 0,C 180,E1 19475.053,E2 19475.053} C_VEL
LIN {X 0,Y 519.649,Z 580.234,A -85,B 0,C 180,E1 19472.012,E2 19472.012} C_VEL
LIN {X 0,Y 518.691,Z 621.19,A -85,B 0,C 180,E1 19468.741,E2 19468.741} C_VEL
LIN {X 0,Y 517.609,Z 660.884,A -85,B 0,C 180,E1 19465.564,E2 19465.564} C_VEL
LIN {X 0,Y 516.331,Z 704.504,A -85,B 0,C 180,E1 19462.066,E2 19462.066} C_VEL
LIN {X 0,Y 516.324,Z 707.916,A -85,B 0,C 180,E1 19461.831,E2 19461.831} C_VEL
LIN {X 0,Y 517.469,Z 718.417,A -85,B 0,C 180,E1 19461.626,E2 19461.626} C_VEL
LIN {X 0,Y 516.343,Z 877.23,A -85,B 0,C 180,E1 19459.334,E2 19459.334} C_VEL
LIN {X 0,Y 516.02,Z 894.369,A -85,B 0,C 180,E1 19458.88,E2 19458.88} C_VEL
LIN {X 0,Y 515.583,Z 910.655,A -85,B 0,C 180,E1 19458.252,E2 19458.252} C_VEL
LIN {X 0,Y 515.036,Z 927.039,A -85,B 0,C 180,E1 19457.396,E2 19457.396} C_VEL
LIN {X 0,Y 514.393,Z 942.931,A -85,B 0,C 180,E1 19456.313,E2 19456.313} C_VEL
LIN {X 0,Y 513.753,Z 958.025,A -85,B 0,C 180,E1 19455.002,E2 19455.002} C_VEL
LIN {X 0,Y 513.18,Z 971.814,A -85,B 0,C 180,E1 19453.521,E2 19453.521} C_VEL
LIN {X 0,Y 512.74,Z 983.013,A -85,B 0,C 180,E1 19452.044,E2 19452.044} C_VEL
LIN {X 0,Y 512.402,Z 993.035,A -85,B 0,C 180,E1 19450.432,E2 19450.432} C_VEL
LIN {X 0,Y 512.144,Z 1002.39,A -85,B 0,C 180,E1 19448.533,E2 19448.533} C_VEL
LIN {X 0,Y 511.998,Z 1009.567,A -85,B 0,C 180,E1 19446.617,E2 19446.617} C_VEL
LIN {X 0,Y 511.935,Z 1014.742,A -85,B 0,C 180,E1 19444.706,E2 19444.706} C_VEL
LIN {X 0,Y 511.917,Z 1018.134,A -85,B 0,C 180,E1 19442.799,E2 19442.799} C_VEL
LIN {X 0,Y 511.915,Z 1019.835,A -85,B 0,C 180,E1 19440.784,E2 19440.784} C_VEL
LIN {X 0,Y 511.916,Z 1019.673,A -85,B 0,C 180,E1 19438.881,E2 19438.881} C_VEL
LIN {X 0,Y 511.915,Z 1017.955,A -85,B 0,C 180,E1 19436.977,E2 19436.977} C_VEL
LIN {X 0,Y 511.944,Z 1014.106,A -85,B 0,C 180,E1 19434.916,E2 19434.916} C_VEL
LIN {X 0,Y 512.02,Z 1008.376,A -85,B 0,C 180,E1 19432.934,E2 19432.934} C_VEL
LIN {X 0,Y 512.164,Z 1001.219,A -85,B 0,C 180,E1 19431.128,E2 19431.128} C_VEL
LIN {X 0,Y 512.388,Z 993.409,A -85,B 0,C 180,E1 19429.545,E2 19429.545} C_VEL
LIN {X 0,Y 512.779,Z 982.094,A -85,B 0,C 180,E1 19427.729,E2 19427.729} C_VEL
LIN {X 0,Y 513.215,Z 970.539,A -85,B 0,C 180,E1 19426.251,E2 19426.251} C_VEL
LIN {X 0,Y 513.653,Z 959.949,A -85,B 0,C 180,E1 19425.111,E2 19425.111} C_VEL
LIN {X 0,Y 514.171,Z 948.313,A -85,B 0,C 180,E1 19424.036,E2 19424.036} C_VEL
LIN {X 0,Y 514.776,Z 933.895,A -85,B 0,C 180,E1 19422.945,E2 19422.945} C_VEL
LIN {X 0,Y 515.324,Z 918.276,A -85,B 0,C 180,E1 19422.032,E2 19422.032} C_VEL
LIN {X 0,Y 515.816,Z 902.417,A -85,B 0,C 180,E1 19421.318,E2 19421.318} C_VEL
LIN {X 0,Y 516.169,Z 885.391,A -85,B 0,C 180,E1 19420.781,E2 19420.781} C_VEL
LIN {X 0,Y 516.38,Z 867.362,A -85,B 0,C 180,E1 19420.429,E2 19420.429} C_VEL
LIN {X 0,Y 517.182,Z 715.125,A -85,B 0,C 180,E1 19418.271,E2 19418.271} C_VEL
LIN {X 0,Y 516.384,Z 708.804,A -85,B 0,C 180,E1 19418.116,E2 19418.116} C_VEL
LIN {X 0,Y 517.44,Z 668.78,A -85,B 0,C 180,E1 19414.965,E2 19414.965} C_VEL
LIN {X 0,Y 518.033,Z 630.788,A -85,B 0,C 180,E1 19412.085,E2 19412.085} C_VEL
LIN {X 0,Y 518.083,Z 595.992,A -85,B 0,C 180,E1 19409.569,E2 19409.569} C_VEL
LIN {X 0,Y 517.644,Z 561.98,A -85,B 0,C 180,E1 19407.26,E2 19407.26} C_VEL
LIN {X 0,Y 516.899,Z 536.017,A -85,B 0,C 180,E1 19405.61,E2 19405.61} C_VEL
LIN {X 0,Y 512.75,Z 520.028,A -85,B 0,C 180,E1 19404.473,E2 19404.473} C_VEL
LIN {X 0,Y 512.605,Z 519.25,A -85,B 0,C 180,E1 19404.324,E2 19404.324} C_VEL
LIN {X 0,Y 512.647,Z 519.154,A -85,B 0,C 180,E1 19400.919,E2 19400.919} C_VEL
LIN {X 0,Y 512.666,Z 519.43,A -85,B 0,C 180,E1 19398.305,E2 19398.305} C_VEL
LIN {X 0,Y 514.176,Z 523.015,A -85,B 0,C 180,E1 19397.715,E2 19397.715} C_VEL
LIN {X 0,Y 521.939,Z 539.521,A -85,B 0,C 180,E1 19395.251,E2 19395.251} C_VEL
LIN {X 0,Y 524.681,Z 545.474,A -85,B 0,C 180,E1 19394.467,E2 19394.467} C_VEL
LIN {X 0,Y 531.547,Z 556.234,A -85,B 0,C 180,E1 19393.608,E2 19393.608} C_VEL
LIN {X 0,Y 533.738,Z 566.799,A -85,B 0,C 180,E1 19393.217,E2 19393.217} C_VEL
LIN {X 0,Y 531.202,Z 752.269,A -85,B 0,C 180,E1 19390.254,E2 19390.254} C_VEL
LIN {X 0,Y 529.052,Z 892.28,A -85,B 0,C 180,E1 19388.01,E2 19388.01} C_VEL
LIN {X 0,Y 528.196,Z 915.215,A -85,B 0,C 180,E1 19387.458,E2 19387.458} C_VEL
LIN {X 0,Y 527.209,Z 935.702,A -85,B 0,C 180,E1 19386.794,E2 19386.794} C_VEL
LIN {X 0,Y 525.86,Z 958.381,A -85,B 0,C 180,E1 19385.847,E2 19385.847} C_VEL
LIN {X 0,Y 524.538,Z 978.573,A -85,B 0,C 180,E1 19384.813,E2 19384.813} C_VEL
LIN {X 0,Y 522.891,Z 1000.133,A -85,B 0,C 180,E1 19383.481,E2 19383.481} C_VEL
LIN {X 0,Y 521.358,Z 1019.971,A -85,B 0,C 180,E1 19382.042,E2 19382.042} C_VEL
LIN {X 0,Y 519.723,Z 1039.267,A -85,B 0,C 180,E1 19380.396,E2 19380.396} C_VEL
LIN {X 0,Y 518.081,Z 1059.138,A -85,B 0,C 180,E1 19378.43,E2 19378.43} C_VEL
LIN {X 0,Y 516.728,Z 1075.658,A -85,B 0,C 180,E1 19376.55,E2 19376.55} C_VEL
LIN {X 0,Y 515.531,Z 1091.144,A -85,B 0,C 180,E1 19374.522,E2 19374.522} C_VEL
LIN {X 0,Y 514.47,Z 1106.22,A -85,B 0,C 180,E1 19372.271,E2 19372.271} C_VEL
LIN {X 0,Y 513.635,Z 1119.089,A -85,B 0,C 180,E1 19370.036,E2 19370.036} C_VEL
LIN {X 0,Y 512.946,Z 1131.805,A -85,B 0,C 180,E1 19367.469,E2 19367.469} C_VEL
LIN {X 0,Y 512.516,Z 1141.529,A -85,B 0,C 180,E1 19365.154,E2 19365.154} C_VEL
LIN {X 0,Y 512.193,Z 1150.345,A -85,B 0,C 180,E1 19362.629,E2 19362.629} C_VEL
LIN {X 0,Y 512.044,Z 1156.866,A -85,B 0,C 180,E1 19360.349,E2 19360.349} C_VEL
LIN {X 0,Y 511.954,Z 1162.635,A -85,B 0,C 180,E1 19357.745,E2 19357.745} C_VEL
LIN {X 0,Y 511.906,Z 1166.277,A -85,B 0,C 180,E1 19355.492,E2 19355.492} C_VEL
LIN {X 0,Y 511.891,Z 1168.919,A -85,B 0,C 180,E1 19352.911,E2 19352.911} C_VEL
LIN {X 0,Y 511.884,Z 1169.872,A -85,B 0,C 180,E1 19350.672,E2 19350.672} C_VEL
LIN {X 0,Y 511.906,Z 1169.526,A -85,B 0,C 180,E1 19348.097,E2 19348.097} C_VEL
LIN {X 0,Y 511.912,Z 1167.616,A -85,B 0,C 180,E1 19345.631,E2 19345.631} C_VEL
LIN {X 0,Y 511.916,Z 1164.081,A -85,B 0,C 180,E1 19343.045,E2 19343.045} C_VEL
LIN {X 0,Y 511.997,Z 1159.573,A -85,B 0,C 180,E1 19340.785,E2 19340.785} C_VEL
LIN {X 0,Y 512.135,Z 1153.175,A -85,B 0,C 180,E1 19338.285,E2 19338.285} C_VEL
LIN {X 0,Y 512.357,Z 1145.343,A -85,B 0,C 180,E1 19335.881,E2 19335.881} C_VEL
LIN {X 0,Y 512.747,Z 1135.938,A -85,B 0,C 180,E1 19333.459,E2 19333.459} C_VEL
LIN {X 0,Y 513.277,Z 1125.152,A -85,B 0,C 180,E1 19331.133,E2 19331.133} C_VEL
LIN {X 0,Y 514.074,Z 1111.858,A -85,B 0,C 180,E1 19328.672,E2 19328.672} C_VEL
LIN {X 0,Y 514.993,Z 1098.565,A -85,B 0,C 180,E1 19326.546,E2 19326.546} C_VEL
LIN {X 0,Y 516.179,Z 1082.725,A -85,B 0,C 180,E1 19324.346,E2 19324.346} C_VEL
LIN {X 0,Y 517.523,Z 1065.989,A -85,B 0,C 180,E1 19322.312,E2 19322.312} C_VEL
LIN {X 0,Y 518.992,Z 1048.176,A -85,B 0,C 180,E1 19320.449,E2 19320.449} C_VEL
LIN {X 0,Y 520.633,Z 1028.259,A -85,B 0,C 180,E1 19318.638,E2 19318.638} C_VEL
LIN {X 0,Y 522.24,Z 1008.897,A -85,B 0,C 180,E1 19317.127,E2 19317.127} C_VEL
LIN {X 0,Y 523.82,Z 987.824,A -85,B 0,C 180,E1 19315.73,E2 19315.73} C_VEL
LIN {X 0,Y 525.41,Z 966.067,A -85,B 0,C 180,E1 19314.52,E2 19314.52} C_VEL
LIN {X 0,Y 526.678,Z 945.2,A -85,B 0,C 180,E1 19313.578,E2 19313.578} C_VEL
LIN {X 0,Y 527.838,Z 923.292,A -85,B 0,C 180,E1 19312.777,E2 19312.777} C_VEL
LIN {X 0,Y 528.732,Z 901.158,A -85,B 0,C 180,E1 19312.18,E2 19312.18} C_VEL
LIN {X 0,Y 529.422,Z 874.675,A -85,B 0,C 180,E1 19311.687,E2 19311.687} C_VEL
LIN {X 0,Y 532.488,Z 664.564,A -85,B 0,C 180,E1 19308.342,E2 19308.342} C_VEL
LIN {X 0,Y 533.664,Z 561.876,A -85,B 0,C 180,E1 19306.689,E2 19306.689} C_VEL
LIN {X 0,Y 532.32,Z 555.476,A -85,B 0,C 180,E1 19306.451,E2 19306.451} C_VEL
LIN {X 0,Y 524.381,Z 543.324,A -85,B 0,C 180,E1 19305.438,E2 19305.438} C_VEL
LIN {X 0,Y 516.675,Z 527.675,A -85,B 0,C 180,E1 19303.392,E2 19303.392} C_VEL
LIN {X 0,Y 513.796,Z 522.458,A -85,B 0,C 180,E1 19302.642,E2 19302.642} C_VEL
LIN {X 0,Y 512.675,Z 519.415,A -85,B 0,C 180,E1 19302.192,E2 19302.192} C_VEL
LIN {X 0,Y 512.636,Z 519.193,A -85,B 0,C 180,E1 19298.902,E2 19298.902} C_VEL
LIN {X 0,Y 512.636,Z 519.186,A -85,B 0,C 180,E1 19295.385,E2 19295.385} C_VEL
LIN {X 0,Y 512.637,Z 519.168,A -85,B 0,C 180,E1 19291.908,E2 19291.908} C_VEL
LIN {X 0,Y 512.641,Z 519.178,A -85,B 0,C 180,E1 19288.401,E2 19288.401} C_VEL
LIN {X 0,Y 512.635,Z 519.192,A -85,B 0,C 180,E1 19284.912,E2 19284.912} C_VEL
LIN {X 0,Y 512.636,Z 519.164,A -85,B 0,C 180,E1 19281.391,E2 19281.391} C_VEL
LIN {X 0,Y 512.64,Z 519.187,A -85,B 0,C 180,E1 19277.831,E2 19277.831} C_VEL
LIN {X 0,Y 512.628,Z 519.171,A -85,B 0,C 180,E1 19274.342,E2 19274.342} C_VEL
LIN {X 0,Y 512.638,Z 519.186,A -85,B 0,C 180,E1 19270.905,E2 19270.905} C_VEL
LIN {X 0,Y 512.645,Z 519.171,A -85,B 0,C 180,E1 19267.283,E2 19267.283} C_VEL
LIN {X 0,Y 512.629,Z 519.183,A -85,B 0,C 180,E1 19263.802,E2 19263.802} C_VEL
LIN {X 0,Y 512.639,Z 519.189,A -85,B 0,C 180,E1 19260.335,E2 19260.335} C_VEL
LIN {X 0,Y 512.642,Z 519.184,A -85,B 0,C 180,E1 19256.745,E2 19256.745} C_VEL
LIN {X 0,Y 512.628,Z 519.184,A -85,B 0,C 180,E1 19253.279,E2 19253.279} C_VEL
LIN {X 0,Y 512.638,Z 519.191,A -85,B 0,C 180,E1 19249.89,E2 19249.89} C_VEL
LIN {X 0,Y 512.641,Z 519.171,A -85,B 0,C 180,E1 19246.349,E2 19246.349} C_VEL
LIN {X 0,Y 512.631,Z 519.183,A -85,B 0,C 180,E1 19242.871,E2 19242.871} C_VEL
LIN {X 0,Y 512.638,Z 519.172,A -85,B 0,C 180,E1 19239.424,E2 19239.424} C_VEL
LIN {X 0,Y 512.626,Z 519.179,A -85,B 0,C 180,E1 19236.065,E2 19236.065} C_VEL
LIN {X 0,Y 512.639,Z 519.189,A -85,B 0,C 180,E1 19232.467,E2 19232.467} C_VEL
LIN {X 0,Y 512.639,Z 519.164,A -85,B 0,C 180,E1 19229.008,E2 19229.008} C_VEL
LIN {X 0,Y 512.623,Z 519.184,A -85,B 0,C 180,E1 19225.553,E2 19225.553} C_VEL
LIN {X 0,Y 512.644,Z 519.194,A -85,B 0,C 180,E1 19221.996,E2 19221.996} C_VEL
LIN {X 0,Y 512.643,Z 519.183,A -85,B 0,C 180,E1 19218.46,E2 19218.46} C_VEL
LIN {X 0,Y 512.663,Z 519.429,A -85,B 0,C 180,E1 19215.426,E2 19215.426} C_VEL
LIN {X 0,Y 512.717,Z 519.742,A -85,B 0,C 180,E1 19215.36,E2 19215.36} C_VEL
LIN {X 0,Y 514.066,Z 527.615,A -85,B 0,C 180,E1 19214.492,E2 19214.492} C_VEL
LIN {X 0,Y 515.624,Z 541.801,A -85,B 0,C 180,E1 19213.105,E2 19213.105} C_VEL
LIN {X 0,Y 516.768,Z 545.52,A -85,B 0,C 180,E1 19212.666,E2 19212.666} C_VEL
LIN {X 0,Y 521.414,Z 556.124,A -85,B 0,C 180,E1 19211.31,E2 19211.31} C_VEL
LIN {X 0,Y 519.555,Z 589.183,A -85,B 0,C 180,E1 19208.893,E2 19208.893} C_VEL
LIN {X 0,Y 522.961,Z 610.529,A -85,B 0,C 180,E1 19208.191,E2 19208.191} C_VEL
LIN {X 0,Y 519.166,Z 842.415,A -85,B 0,C 180,E1 19204.506,E2 19204.506} C_VEL
LIN {X 0,Y 518.326,Z 897.416,A -85,B 0,C 180,E1 19203.625,E2 19203.625} C_VEL
LIN {X 0,Y 517.504,Z 918.675,A -85,B 0,C 180,E1 19203.089,E2 19203.089} C_VEL
LIN {X 0,Y 516.477,Z 940.435,A -85,B 0,C 180,E1 19202.33,E2 19202.33} C_VEL
LIN {X 0,Y 515.318,Z 960.71,A -85,B 0,C 180,E1 19201.426,E2 19201.426} C_VEL
LIN {X 0,Y 513.946,Z 980.549,A -85,B 0,C 180,E1 19200.321,E2 19200.321} C_VEL
LIN {X 0,Y 512.528,Z 1000.242,A -85,B 0,C 180,E1 19198.998,E2 19198.998} C_VEL
LIN {X 0,Y 511.126,Z 1018.447,A -85,B 0,C 180,E1 19197.558,E2 19197.558} C_VEL
LIN {X 0,Y 509.693,Z 1036.251,A -85,B 0,C 180,E1 19195.892,E2 19195.892} C_VEL
LIN {X 0,Y 508.382,Z 1052.797,A -85,B 0,C 180,E1 19194.086,E2 19194.086} C_VEL
LIN {X 0,Y 507.205,Z 1068.361,A -85,B 0,C 180,E1 19192.118,E2 19192.118} C_VEL
LIN {X 0,Y 506.196,Z 1082.848,A -85,B 0,C 180,E1 19189.982,E2 19189.982} C_VEL
LIN {X 0,Y 505.415,Z 1095.079,A -85,B 0,C 180,E1 19187.857,E2 19187.857} C_VEL
LIN {X 0,Y 504.805,Z 1106.603,A -85,B 0,C 180,E1 19185.509,E2 19185.509} C_VEL
LIN {X 0,Y 504.403,Z 1116.192,A -85,B 0,C 180,E1 19183.177,E2 19183.177} C_VEL
LIN {X 0,Y 504.146,Z 1123.89,A -85,B 0,C 180,E1 19180.86,E2 19180.86} C_VEL
LIN {X 0,Y 503.995,Z 1130.546,A -85,B 0,C 180,E1 19178.327,E2 19178.327} C_VEL
LIN {X 0,Y 503.93,Z 1135.254,A -85,B 0,C 180,E1 19175.922,E2 19175.922} C_VEL
LIN {X 0,Y 503.908,Z 1138.242,A -85,B 0,C 180,E1 19173.527,E2 19173.527} C_VEL
LIN {X 0,Y 503.908,Z 1139.793,A -85,B 0,C 180,E1 19171.023,E2 19171.023} C_VEL
LIN {X 0,Y 503.906,Z 1139.745,A -85,B 0,C 180,E1 19168.636,E2 19168.636} C_VEL
LIN {X 0,Y 503.907,Z 1138.106,A -85,B 0,C 180,E1 19166.246,E2 19166.246} C_VEL
LIN {X 0,Y 503.935,Z 1135.01,A -85,B 0,C 180,E1 19163.849,E2 19163.849} C_VEL
LIN {X 0,Y 504.004,Z 1130.236,A -85,B 0,C 180,E1 19161.443,E2 19161.443} C_VEL
LIN {X 0,Y 504.147,Z 1123.812,A -85,B 0,C 180,E1 19159.024,E2 19159.024} C_VEL
LIN {X 0,Y 504.408,Z 1116.097,A -85,B 0,C 180,E1 19156.706,E2 19156.706} C_VEL
LIN {X 0,Y 504.817,Z 1106.48,A -85,B 0,C 180,E1 19154.373,E2 19154.373} C_VEL
LIN {X 0,Y 505.425,Z 1094.926,A -85,B 0,C 180,E1 19152.025,E2 19152.025} C_VEL
LIN {X 0,Y 506.208,Z 1082.655,A -85,B 0,C 180,E1 19149.898,E2 19149.898} C_VEL
LIN {X 0,Y 507.221,Z 1068.134,A -85,B 0,C 180,E1 19147.76,E2 19147.76} C_VEL
LIN {X 0,Y 508.404,Z 1052.524,A -85,B 0,C 180,E1 19145.792,E2 19145.792} C_VEL
LIN {X 0,Y 509.76,Z 1035.427,A -85,B 0,C 180,E1 19143.937,E2 19143.937} C_VEL
LIN {X 0,Y 511.204,Z 1017.34,A -85,B 0,C 180,E1 19142.257,E2 19142.257} C_VEL
LIN {X 0,Y 512.634,Z 998.948,A -85,B 0,C 180,E1 19140.816,E2 19140.816} C_VEL
LIN {X 0,Y 514.054,Z 978.937,A -85,B 0,C 180,E1 19139.492,E2 19139.492} C_VEL
LIN {X 0,Y 515.44,Z 958.651,A -85,B 0,C 180,E1 19138.384,E2 19138.384} C_VEL
LIN {X 0,Y 516.566,Z 938.758,A -85,B 0,C 180,E1 19137.512,E2 19137.512} C_VEL
LIN {X 0,Y 517.568,Z 917.251,A -85,B 0,C 180,E1 19136.781,E2 19136.781} C_VEL
LIN {X 0,Y 518.36,Z 895.98,A -85,B 0,C 180,E1 19136.257,E2 19136.257} C_VEL
LIN {X 0,Y 522.129,Z 659.746,A -85,B 0,C 180,E1 19132.507,E2 19132.507} C_VEL
LIN {X 0,Y 522.737,Z 611.525,A -85,B 0,C 180,E1 19131.715,E2 19131.715} C_VEL
LIN {X 0,Y 518.142,Z 589.012,A -85,B 0,C 180,E1 19130.839,E2 19130.839} C_VEL
LIN {X 0,Y 520.25,Z 556.031,A -85,B 0,C 180,E1 19127.876,E2 19127.876} C_VEL
LIN {X 0,Y 513.317,Z 539.584,A -85,B 0,C 180,E1 19125.472,E2 19125.472} C_VEL
LIN {X 0,Y 506.204,Z 523.919,A -85,B 0,C 180,E1 19122.957,E2 19122.957} C_VEL
LIN {X 0,Y 504.675,Z 520.374,A -85,B 0,C 180,E1 19122.311,E2 19122.311} C_VEL
LIN {X 0,Y 504.671,Z 520.185,A -85,B 0,C 180,E1 19119.492,E2 19119.492} C_VEL
LIN {X 0,Y 504.679,Z 520.419,A -85,B 0,C 180,E1 19117.908,E2 19117.908} C_VEL
LIN {X 0,Y 511.692,Z 540.52,A -85,B 0,C 180,E1 19115.751,E2 19115.751} C_VEL
LIN {X 0,Y 513.068,Z 545.751,A -85,B 0,C 180,E1 19115.229,E2 19115.229} C_VEL
LIN {X 0,Y 512.264,Z 586.752,A -85,B 0,C 180,E1 19111.935,E2 19111.935} C_VEL
LIN {X 0,Y 511.189,Z 627.785,A -85,B 0,C 180,E1 19108.634,E2 19108.634} C_VEL
LIN {X 0,Y 509.938,Z 671.535,A -85,B 0,C 180,E1 19105.113,E2 19105.113} C_VEL
LIN {X 0,Y 508.826,Z 708.726,A -85,B 0,C 180,E1 19102.142,E2 19102.142} C_VEL
LIN {X 0,Y 509.973,Z 719.181,A -85,B 0,C 180,E1 19101.93,E2 19101.93} C_VEL
LIN {X 0,Y 508.694,Z 878.448,A -85,B 0,C 180,E1 19099.58,E2 19099.58} C_VEL
LIN {X 0,Y 508.369,Z 895.91,A -85,B 0,C 180,E1 19099.112,E2 19099.112} C_VEL
LIN {X 0,Y 507.878,Z 913.183,A -85,B 0,C 180,E1 19098.42,E2 19098.42} C_VEL
LIN {X 0,Y 507.321,Z 929.28,A -85,B 0,C 180,E1 19097.55,E2 19097.55} C_VEL
LIN {X 0,Y 506.688,Z 944.238,A -85,B 0,C 180,E1 19096.509,E2 19096.509} C_VEL
LIN {X 0,Y 506.04,Z 958.725,A -85,B 0,C 180,E1 19095.236,E2 19095.236} C_VEL
LIN {X 0,Y 505.436,Z 971.455,A -85,B 0,C 180,E1 19093.849,E2 19093.849} C_VEL
LIN {X 0,Y 504.913,Z 982.655,A -85,B 0,C 180,E1 19092.349,E2 19092.349} C_VEL
LIN {X 0,Y 504.475,Z 993.036,A -85,B 0,C 180,E1 19090.622,E2 19090.622} C_VEL
LIN {X 0,Y 504.173,Z 1002.393,A -85,B 0,C 180,E1 19088.669,E2 19088.669} C_VEL
LIN {X 0,Y 504.011,Z 1009.567,A -85,B 0,C 180,E1 19086.722,E2 19086.722} C_VEL
LIN {X 0,Y 503.938,Z 1014.744,A -85,B 0,C 180,E1 19084.78,E2 19084.78} C_VEL
LIN {X 0,Y 503.917,Z 1018.133,A -85,B 0,C 180,E1 19082.844,E2 19082.844} C_VEL
LIN {X 0,Y 503.915,Z 1019.834,A -85,B 0,C 180,E1 19080.796,E2 19080.796} C_VEL
LIN {X 0,Y 503.916,Z 1019.666,A -85,B 0,C 180,E1 19078.863,E2 19078.863} C_VEL
LIN {X 0,Y 503.916,Z 1017.954,A -85,B 0,C 180,E1 19076.929,E2 19076.929} C_VEL
LIN {X 0,Y 503.949,Z 1014.188,A -85,B 0,C 180,E1 19074.872,E2 19074.872} C_VEL
LIN {X 0,Y 504.025,Z 1008.719,A -85,B 0,C 180,E1 19072.936,E2 19072.936} C_VEL
LIN {X 0,Y 504.199,Z 1001.112,A -85,B 0,C 180,E1 19070.957,E2 19070.957} C_VEL
LIN {X 0,Y 504.538,Z 991.723,A -85,B 0,C 180,E1 19069.033,E2 19069.033} C_VEL
LIN {X 0,Y 505.017,Z 981.04,A -85,B 0,C 180,E1 19067.305,E2 19067.305} C_VEL
LIN {X 0,Y 505.52,Z 970.434,A -85,B 0,C 180,E1 19065.92,E2 19065.92} C_VEL
LIN {X 0,Y 506.122,Z 958.134,A -85,B 0,C 180,E1 19064.593,E2 19064.593} C_VEL
LIN {X 0,Y 506.734,Z 944.123,A -85,B 0,C 180,E1 19063.375,E2 19063.375} C_VEL
LIN {X 0,Y 507.317,Z 929.89,A -85,B 0,C 180,E1 19062.391,E2 19062.391} C_VEL
LIN {X 0,Y 507.848,Z 913.716,A -85,B 0,C 180,E1 19061.52,E2 19061.52} C_VEL
LIN {X 0,Y 508.291,Z 896.819,A -85,B 0,C 180,E1 19060.848,E2 19060.848} C_VEL
LIN {X 0,Y 508.576,Z 879.628,A -85,B 0,C 180,E1 19060.393,E2 19060.393} C_VEL
LIN {X 0,Y 509.593,Z 715.95,A -85,B 0,C 180,E1 19057.994,E2 19057.994} C_VEL
LIN {X 0,Y 508.984,Z 710.63,A -85,B 0,C 180,E1 19057.842,E2 19057.842} C_VEL
LIN {X 0,Y 510.008,Z 670.002,A -85,B 0,C 180,E1 19054.66,E2 19054.66} C_VEL
LIN {X 0,Y 510.548,Z 634.388,A -85,B 0,C 180,E1 19051.965,E2 19051.965} C_VEL
LIN {X 0,Y 510.607,Z 598.799,A -85,B 0,C 180,E1 19049.395,E2 19049.395} C_VEL
LIN {X 0,Y 510.137,Z 564.476,A -85,B 0,C 180,E1 19047.071,E2 19047.071} C_VEL
